C07209=1031.022,-23.750,-88.174,168.001,42.640,157.928
C07210=1031.029,-23.500,-88.188,168.003,42.639,157.928
C07211=1031.035,-23.251,-88.201,168.006,42.638,157.928
C07212=1031.041,-23.002,-88.215,168.009,42.636,157.928
C07213=1031.047,-22.752,-88.229,168.012,42.635,157.928
C07214=1031.053,-22.502,-88.242,168.014,42.634,157.928
C07215=1031.060,-22.253,-88.255,168.016,42.633,157.928
C07216=1031.066,-22.003,-88.270,168.019,42.631,157.928
C07217=1031.072,-21.754,-88.283,168.022,42.630,157.928
C07218=1031.078,-21.504,-88.296,168.025,42.629,157.928
C07219=1031.084,-21.254,-88.310,168.026,42.627,157.928
C07220=1031.091,-21.005,-88.324,168.029,42.626,157.928
C07221=1031.097,-20.756,-88.338,168.032,42.625,157.928
C07222=1031.104,-20.474,-88.353,168.035,42.623,157.928
C07223=1031.111,-20.193,-88.369,168.038,42.622,157.928
C07224=1031.118,-19.911,-88.384,168.040,42.621,157.928
C07225=1031.125,-19.630,-88.399,168.043,42.619,157.928
C07226=1031.131,-19.380,-88.413,168.046,42.618,157.928
C07227=1031.138,-19.130,-88.426,168.049,42.617,157.928
C07228=1031.145,-18.881,-88.441,168.051,42.615,157.927
C07229=1031.150,-18.632,-88.455,168.053,42.614,157.927
C07230=1031.156,-18.382,-88.468,168.056,42.613,157.927
C07231=1031.163,-18.132,-88.481,168.059,42.611,157.927
C07232=1031.169,-17.883,-88.495,168.061,42.610,157.927
C07233=1031.176,-17.633,-88.510,168.064,42.609,157.927
C07234=1031.182,-17.384,-88.523,168.066,42.608,157.927
C07235=1031.188,-17.134,-88.537,168.069,42.606,157.927
C07236=1031.194,-16.885,-88.550,168.071,42.605,157.927
C07237=1031.200,-16.635,-88.564,168.074,42.604,157.927
C07238=1031.207,-16.386,-88.579,168.077,42.602,157.927
C07239=1031.213,-16.136,-88.592,168.079,42.601,157.927
C07240=1031.220,-15.886,-88.606,168.081,42.600,157.927
C07241=1031.226,-15.638,-88.620,168.084,42.598,157.927
C07242=1031.232,-15.388,-88.634,168.087,42.597,157.927
C07243=1031.238,-15.138,-88.648,168.090,42.596,157.927
C07244=1031.245,-14.889,-88.662,168.091,42.595,157.927
C07245=1031.251,-14.639,-88.676,168.094,42.594,157.927
C07246=1031.257,-14.389,-88.690,168.097,42.592,157.927
C07247=1031.263,-14.140,-88.704,168.099,42.591,157.926
C07248=1031.269,-13.890,-88.718,168.102,42.590,157.926
C07249=1031.275,-13.641,-88.732,168.105,42.589,157.926
C07250=1031.282,-13.391,-88.747,168.106,42.588,157.926
C07251=1031.288,-13.142,-88.760,168.109,42.586,157.926
C07252=1031.294,-12.892,-88.775,168.112,42.585,157.926
C07253=1031.300,-12.642,-88.789,168.114,42.584,157.926
C07254=1031.307,-12.393,-88.803,168.117,42.583,157.926
C07255=1031.313,-12.144,-88.817,168.119,42.581,157.926
C07256=1031.319,-11.894,-88.830,168.121,42.580,157.926
C07257=1031.325,-11.645,-88.845,168.124,42.579,157.926
C07258=1031.332,-11.395,-88.859,168.127,42.578,157.926
C07259=1031.338,-11.146,-88.873,168.130,42.576,157.926
C07260=1031.344,-10.895,-88.888,168.132,42.575,157.926
C07261=1031.350,-10.647,-88.901,168.134,42.574,157.926
C07262=1031.356,-10.396,-88.916,168.137,42.573,157.926
C07263=1031.363,-10.148,-88.930,168.139,42.572,157.926
C07264=1031.369,-9.898,-88.944,168.142,42.570,157.926
C07265=1031.375,-9.648,-88.959,168.145,42.569,157.926
C07266=1031.382,-9.399,-88.972,168.146,42.568,157.926
C07267=1031.388,-9.149,-88.987,168.149,42.567,157.926
C07268=1031.394,-8.900,-89.002,168.152,42.566,157.926
C07269=1031.401,-8.650,-89.015,168.154,42.564,157.925
C07270=1031.406,-8.401,-89.030,168.157,42.563,157.925
C07271=1031.413,-8.151,-89.044,168.160,42.562,157.925
C07272=1031.420,-7.901,-89.058,168.161,42.561,157.925
C07273=1031.425,-7.652,-89.072,168.164,42.559,157.925
C07274=1031.432,-7.403,-89.087,168.167,42.558,157.925
C07275=1031.438,-7.154,-89.101,168.169,42.557,157.925
C07276=1031.445,-6.904,-89.115,168.172,42.556,157.925
C07277=1031.451,-6.654,-89.130,168.175,42.555,157.925
C07278=1031.457,-6.404,-89.144,168.176,42.553,157.925
C07279=1031.464,-6.155,-89.158,168.179,42.552,157.925
C07280=1031.470,-5.905,-89.173,168.182,42.551,157.925
C07281=1031.476,-5.656,-89.187,168.184,42.550,157.925
C07282=1031.483,-5.406,-89.201,168.186,42.548,157.925
C07283=1031.489,-5.157,-89.216,168.189,42.547,157.925
C07284=1031.495,-4.908,-89.229,168.191,42.546,157.925
C07285=1031.502,-4.658,-89.244,168.194,42.545,157.925
C07286=1031.509,-4.374,-89.261,168.197,42.543,157.925
C07287=1031.516,-4.092,-89.277,168.199,42.542,157.925
C07288=1031.523,-3.809,-89.293,168.202,42.540,157.924
C07289=1031.530,-3.526,-89.310,168.205,42.539,157.924
C07290=1031.537,-3.276,-89.325,168.208,42.538,157.924
C07291=1031.543,-3.027,-89.339,168.210,42.537,157.924
C07292=1031.549,-2.777,-89.354,168.213,42.536,157.924
C07293=1031.555,-2.528,-89.369,168.215,42.535,157.924
C07294=1031.561,-2.278,-89.383,168.217,42.534,157.924
C07295=1031.567,-2.028,-89.398,168.220,42.533,157.924
C07296=1031.574,-1.779,-89.413,168.222,42.532,157.924
C07297=1031.579,-1.530,-89.427,168.225,42.531,157.924
C07298=1031.586,-1.280,-89.442,168.227,42.530,157.924
C07299=1031.592,-1.031,-89.457,168.230,42.529,157.924
C07300=1031.598,-0.782,-89.472,168.232,42.527,157.924
C07301=1031.604,-0.532,-89.487,168.234,42.527,157.924
C07302=1031.610,-0.282,-89.501,168.237,42.525,157.924
C07303=1031.616,-0.033,-89.516,168.239,42.524,157.924
C07304=1031.623,0.217,-89.530,168.242,42.523,157.924
C07305=1031.629,0.467,-89.545,168.245,42.522,157.924
C07306=1031.635,0.716,-89.560,168.246,42.521,157.924
C07307=1031.641,0.965,-89.575,168.249,42.519,157.924
C07308=1031.647,1.215,-89.590,168.251,42.518,157.924
C07309=1031.654,1.465,-89.605,168.254,42.517,157.924
C07310=1031.660,1.713,-89.619,168.257,42.516,157.924
C07311=1031.666,1.963,-89.634,168.259,42.515,157.924
C07312=1031.672,2.213,-89.649,168.261,42.514,157.924
C07313=1031.679,2.462,-89.664,168.263,42.513,157.924
C07314=1031.685,2.711,-89.679,168.266,42.512,157.924
C07315=1031.691,2.961,-89.694,168.268,42.511,157.924
C07316=1031.697,3.211,-89.709,168.271,42.510,157.924
C07317=1031.704,3.460,-89.724,168.274,42.509,157.924
C07318=1031.710,3.709,-89.738,168.275,42.507,157.923
C07319=1031.716,3.959,-89.753,168.278,42.506,157.923
C07320=1031.722,4.209,-89.768,168.280,42.505,157.923
C07321=1031.729,4.458,-89.783,168.283,42.504,157.923
C07322=1031.734,4.707,-89.798,168.286,42.503,157.923
C07323=1031.741,4.957,-89.813,168.288,42.502,157.923
C07324=1031.747,5.207,-89.828,168.290,42.501,157.923
C07325=1031.754,5.456,-89.843,168.292,42.500,157.923
C07326=1031.760,5.706,-89.857,168.295,42.499,157.923
C07327=1031.766,5.956,-89.872,168.298,42.497,157.923
C07328=1031.772,6.204,-89.888,168.300,42.496,157.923
C07329=1031.779,6.454,-89.903,168.303,42.495,157.923
C07330=1031.785,6.703,-89.918,168.304,42.494,157.923
C07331=1031.792,6.953,-89.933,168.307,42.493,157.923
C07332=1031.798,7.203,-89.947,168.309,42.492,157.923
C07333=1031.804,7.452,-89.962,168.312,42.491,157.923
C07334=1031.810,7.701,-89.977,168.315,42.489,157.923
C07335=1031.817,7.951,-89.992,168.316,42.488,157.923
C07336=1031.823,8.200,-90.008,168.319,42.487,157.923
C07337=1031.830,8.449,-90.023,168.321,42.486,157.923
C07338=1031.836,8.699,-90.038,168.324,42.485,157.923
C07339=1031.842,8.949,-90.052,168.327,42.483,157.923
C07340=1031.849,9.198,-90.067,168.329,42.482,157.923
C07341=1031.855,9.447,-90.083,168.332,42.481,157.923
C07342=1031.861,9.696,-90.098,168.333,42.480,157.922
C07343=1031.868,9.946,-90.113,168.336,42.479,157.922
C07344=1031.874,10.196,-90.128,168.338,42.478,157.922
C07345=1031.880,10.445,-90.142,168.341,42.477,157.922
C07346=1031.887,10.694,-90.158,168.344,42.475,157.922
C07347=1031.893,10.944,-90.173,168.345,42.474,157.922
C07348=1031.900,11.194,-90.188,168.348,42.473,157.922
C07349=1031.906,11.443,-90.203,168.350,42.472,157.922
C07350=1031.913,11.728,-90.220,168.353,42.471,157.922
C07351=1031.921,12.013,-90.238,168.356,42.469,157.922
C07352=1031.928,12.298,-90.256,168.358,42.468,157.922
C07353=1031.935,12.583,-90.272,168.361,42.467,157.922
C07354=1031.942,12.833,-90.288,168.364,42.465,157.922
C07355=1031.948,13.082,-90.303,168.366,42.464,157.922
C07356=1031.954,13.332,-90.318,168.369,42.463,157.922
C07357=1031.961,13.581,-90.333,168.370,42.462,157.922
C07358=1031.967,13.831,-90.348,168.373,42.461,157.922
C07359=1031.974,14.080,-90.363,168.376,42.459,157.922
C07360=1031.980,14.330,-90.380,168.378,42.458,157.922
C07361=1031.986,14.579,-90.395,168.381,42.457,157.922
C07362=1031.993,14.828,-90.410,168.383,42.456,157.922
C07363=1031.998,15.078,-90.426,168.386,42.455,157.922
C07364=1032.005,15.328,-90.441,168.387,42.454,157.922
C07365=1032.012,15.577,-90.456,168.390,42.453,157.921
C07366=1032.017,15.827,-90.472,168.392,42.452,157.921
C07367=1032.024,16.076,-90.488,168.395,42.451,157.921
C07368=1032.030,16.326,-90.503,168.397,42.450,157.921
C07369=1032.037,16.575,-90.518,168.400,42.448,157.921
C07370=1032.043,16.825,-90.534,168.401,42.447,157.921
C07371=1032.049,17.073,-90.549,168.404,42.446,157.921
C07372=1032.055,17.323,-90.564,168.406,42.445,157.921
C07373=1032.061,17.572,-90.580,168.409,42.444,157.921
C07374=1032.067,17.822,-90.595,168.411,42.443,157.921
C07375=1032.074,18.071,-90.611,168.414,42.442,157.921
C07376=1032.080,18.321,-90.627,168.415,42.441,157.921
C07377=1032.087,18.570,-90.642,168.418,42.440,157.921
C07378=1032.093,18.820,-90.657,168.420,42.439,157.921
C07379=1032.099,19.069,-90.674,168.423,42.438,157.921
C07380=1032.106,19.319,-90.689,168.426,42.437,157.921
C07381=1032.112,19.568,-90.704,168.428,42.436,157.921
C07382=1032.118,19.817,-90.720,168.431,42.435,157.921
C07383=1032.125,20.067,-90.735,168.432,42.434,157.921
C07384=1032.131,20.316,-90.752,168.435,42.433,157.921
C07385=1032.137,20.566,-90.767,168.437,42.432,157.921
C07386=1032.143,20.815,-90.783,168.440,42.431,157.921
C07387=1032.150,21.064,-90.799,168.442,42.430,157.921
C07388=1032.156,21.314,-90.813,168.445,42.428,157.921
C07389=1032.162,21.563,-90.830,168.446,42.427,157.920
C07390=1032.169,21.812,-90.845,168.448,42.426,157.920
C07391=1032.174,22.062,-90.861,168.451,42.425,157.920
C07392=1032.181,22.311,-90.877,168.453,42.424,157.920
C07393=1032.187,22.561,-90.893,168.456,42.423,157.920
C07394=1032.193,22.810,-90.908,168.458,42.422,157.920
C07395=1032.199,23.060,-90.924,168.460,42.421,157.920
C07396=1032.206,23.309,-90.940,168.462,42.420,157.920
C07397=1032.213,23.559,-90.956,168.465,42.418,157.920
C07398=1032.219,23.809,-90.971,168.467,42.418,157.920
C07399=1032.225,24.058,-90.988,168.470,42.416,157.920
C07400=1032.232,24.307,-91.003,168.472,42.415,157.920
C07401=1032.237,24.557,-91.019,168.475,42.414,157.920
C07402=1032.244,24.806,-91.034,168.476,42.413,157.920
C07403=1032.250,25.055,-91.051,168.479,42.412,157.920
C07404=1032.257,25.304,-91.066,168.481,42.411,157.920
C07405=1032.263,25.554,-91.083,168.484,42.410,157.920
C07406=1032.270,25.804,-91.098,168.486,42.409,157.920
C07407=1032.275,26.053,-91.114,168.489,42.408,157.920
C07408=1032.282,26.302,-91.130,168.490,42.407,157.920
C07409=1032.288,26.552,-91.146,168.493,42.406,157.920
C07410=1032.295,26.801,-91.162,168.495,42.405,157.920
C07411=1032.300,27.051,-91.177,168.498,42.404,157.920
C07412=1032.307,27.300,-91.193,168.500,42.403,157.920
C07413=1032.314,27.550,-91.210,168.503,42.401,157.920
C07414=1032.320,27.835,-91.228,168.505,42.400,157.920
C07415=1032.328,28.122,-91.246,168.507,42.399,157.919
C07416=1032.335,28.409,-91.264,168.510,42.398,157.919
C07417=1032.342,28.695,-91.283,168.513,42.397,157.919
C07418=1032.348,28.944,-91.299,168.516,42.396,157.919
C07419=1032.355,29.193,-91.315,168.518,42.395,157.919
C07420=1032.361,29.442,-91.331,168.520,42.394,157.919
C07421=1032.367,29.692,-91.347,168.522,42.393,157.919
C07422=1032.374,29.942,-91.364,168.524,42.392,157.919
C07423=1032.380,30.191,-91.380,168.527,42.391,157.919
C07424=1032.386,30.440,-91.396,168.529,42.390,157.919
C07425=1032.392,30.690,-91.412,168.532,42.389,157.919
C07426=1032.399,30.939,-91.428,168.534,42.388,157.919
C07427=1032.405,31.189,-91.445,168.536,42.386,157.919
C07428=1032.411,31.438,-91.461,168.538,42.386,157.919
C07429=1032.418,31.687,-91.476,168.540,42.385,157.919
C07430=1032.424,31.936,-91.493,168.543,42.383,157.919
C07431=1032.430,32.186,-91.509,168.545,42.382,157.919
C07432=1032.436,32.436,-91.526,168.548,42.381,157.919
C07433=1032.443,32.685,-91.541,168.550,42.380,157.919
C07434=1032.449,32.934,-91.558,168.552,42.379,157.919
C07435=1032.455,33.184,-91.574,168.554,42.378,157.919
C07436=1032.461,33.433,-91.590,168.557,42.377,157.919
C07437=1032.468,33.683,-91.606,168.559,42.376,157.919
C07438=1032.474,33.932,-91.622,168.562,42.375,157.919
C07439=1032.480,34.181,-91.639,168.564,42.374,157.919
C07440=1032.487,34.430,-91.654,168.566,42.373,157.919
C07441=1032.493,34.680,-91.671,168.568,42.372,157.919
C07442=1032.499,34.930,-91.687,168.570,42.371,157.919
C07443=1032.506,35.179,-91.704,168.573,42.370,157.919
C07444=1032.512,35.428,-91.720,168.575,42.369,157.918
C07445=1032.519,35.678,-91.736,168.578,42.368,157.918
C07446=1032.525,35.927,-91.753,168.580,42.367,157.918
C07447=1032.531,36.176,-91.769,168.582,42.366,157.918
C07448=1032.538,36.426,-91.785,168.584,42.365,157.918
C07449=1032.544,36.675,-91.801,168.587,42.364,157.918
C07450=1032.550,36.924,-91.818,168.589,42.363,157.918
C07451=1032.556,37.173,-91.834,168.591,42.362,157.918
C07452=1032.563,37.424,-91.851,168.594,42.361,157.918
C07453=1032.569,37.673,-91.867,168.596,42.360,157.918
C07454=1032.575,37.922,-91.884,168.598,42.359,157.918
C07455=1032.581,38.172,-91.901,168.600,42.358,157.918
C07456=1032.587,38.421,-91.917,168.603,42.357,157.918
C07457=1032.593,38.670,-91.933,168.605,42.356,157.918
C07458=1032.599,38.920,-91.950,168.607,42.355,157.918
C07459=1032.607,39.169,-91.966,168.610,42.354,157.918
C07460=1032.613,39.418,-91.983,168.612,42.353,157.918
C07461=1032.619,39.668,-91.999,168.615,42.352,157.918
C07462=1032.626,39.917,-92.016,168.616,42.351,157.918
C07463=1032.632,40.166,-92.033,168.618,42.350,157.918
C07464=1032.638,40.416,-92.049,168.621,42.349,157.918
C07465=1032.644,40.665,-92.066,168.623,42.348,157.918
C07466=1032.653,41.053,-92.091,168.627,42.347,157.918
C07467=1032.663,41.442,-92.117,168.631,42.345,157.918
C07468=1032.673,41.830,-92.144,168.634,42.344,157.918
C07469=1032.684,42.219,-92.169,168.637,42.342,157.918
C07470=1032.690,42.467,-92.186,168.640,42.341,157.918
C07471=1032.696,42.717,-92.203,168.642,42.340,157.918
C07472=1032.702,42.967,-92.219,168.645,42.339,157.918
C07473=1032.708,43.216,-92.237,168.646,42.338,157.917
C07474=1032.717,43.613,-92.263,168.650,42.337,157.918
C07475=1032.727,44.009,-92.290,168.653,42.335,157.917
C07476=1032.737,44.406,-92.317,168.657,42.334,157.918
C07477=1032.747,44.803,-92.344,168.661,42.332,157.917
C07478=1032.753,45.051,-92.361,168.663,42.331,157.917
C07479=1032.760,45.301,-92.377,168.666,42.331,157.917
C07480=1032.765,45.550,-92.395,168.667,42.330,157.917
C07481=1032.772,45.800,-92.412,168.669,42.329,157.917
C07482=1032.778,46.049,-92.429,168.672,42.328,157.917
C07483=1032.784,46.298,-92.445,168.674,42.327,157.917
C07484=1032.790,46.548,-92.463,168.677,42.326,157.917
C07485=1032.796,46.798,-92.479,168.679,42.326,157.917
C07486=1032.802,47.046,-92.496,168.681,42.325,157.917
C07487=1032.809,47.296,-92.513,168.684,42.323,157.917
C07488=1032.814,47.545,-92.530,168.685,42.322,157.917
C07489=1032.821,47.795,-92.548,168.687,42.322,157.917
C07490=1032.827,48.044,-92.564,168.690,42.320,157.917
C07491=1032.834,48.294,-92.581,168.692,42.319,157.917
C07492=1032.839,48.543,-92.599,168.695,42.319,157.917
C07493=1032.845,48.792,-92.615,168.697,42.318,157.917
C07494=1032.852,49.041,-92.632,168.699,42.317,157.917
C07495=1032.858,49.290,-92.650,168.702,42.316,157.917
C07496=1032.864,49.541,-92.667,168.703,42.315,157.917
C07497=1032.871,49.789,-92.684,168.705,42.314,157.917
C07498=1032.877,50.039,-92.701,168.708,42.313,157.917
C07499=1032.883,50.288,-92.718,168.710,42.313,157.917
C07500=1032.889,50.537,-92.735,168.713,42.312,157.917
C07501=1032.896,50.786,-92.752,168.715,42.311,157.917
C07502=1032.902,51.036,-92.768,168.717,42.310,157.917
C07503=1032.908,51.286,-92.786,168.720,42.309,157.917
C07504=1032.914,51.534,-92.803,168.721,42.308,157.917
C07505=1032.921,51.784,-92.820,168.724,42.306,157.917
C07506=1032.926,52.033,-92.837,168.726,42.306,157.917
C07507=1032.933,52.283,-92.855,168.728,42.305,157.917
C07508=1032.939,52.532,-92.872,168.731,42.303,157.917
C07509=1032.946,52.782,-92.888,168.733,42.303,157.917
C07510=1032.951,53.031,-92.906,168.735,42.302,157.917
C07511=1032.958,53.280,-92.923,168.738,42.301,157.917
C07512=1032.964,53.529,-92.940,168.739,42.300,157.917
C07513=1032.970,53.779,-92.957,168.742,42.299,157.917
C07514=1032.977,54.028,-92.974,168.744,42.298,157.917
C07515=1032.983,54.277,-92.992,168.746,42.297,157.917
C07516=1032.989,54.526,-93.009,168.749,42.296,157.916
C07517=1032.996,54.776,-93.027,168.751,42.295,157.916
C07518=1033.002,55.026,-93.043,168.753,42.294,157.916
C07519=1033.009,55.275,-93.060,168.755,42.293,157.916
C07520=1033.015,55.524,-93.078,168.757,42.292,157.916
C07521=1033.021,55.773,-93.095,168.760,42.291,157.916
C07522=1033.028,56.022,-93.112,168.762,42.290,157.916
C07523=1033.033,56.272,-93.129,168.765,42.290,157.916
C07524=1033.040,56.522,-93.147,168.767,42.289,157.916
C07525=1033.047,56.771,-93.164,168.769,42.288,157.916
C07526=1033.052,57.020,-93.182,168.771,42.287,157.916
C07527=1033.059,57.269,-93.199,168.773,42.286,157.916
C07528=1033.065,57.518,-93.216,168.776,42.284,157.916
C07529=1033.071,57.768,-93.234,168.778,42.284,157.916
C07530=1033.078,58.017,-93.251,168.780,42.283,157.916
C07531=1033.084,58.267,-93.267,168.783,42.281,157.916
C07532=1033.090,58.516,-93.285,168.785,42.280,157.916
C07533=1033.097,58.765,-93.302,168.787,42.279,157.916
C07534=1033.104,59.015,-93.320,168.789,42.278,157.916
C07535=1033.110,59.264,-93.338,168.791,42.277,157.916
C07536=1033.116,59.513,-93.355,168.794,42.276,157.916
C07537=1033.123,59.763,-93.372,168.796,42.275,157.916
C07538=1033.130,60.048,-93.392,168.799,42.274,157.916
C07539=1033.137,60.334,-93.412,168.802,42.273,157.916
C07540=1033.144,60.620,-93.431,168.803,42.272,157.916
C07541=1033.152,60.907,-93.451,168.806,42.270,157.915
C07542=1033.158,61.155,-93.468,168.809,42.269,157.915
C07543=1033.164,61.405,-93.486,168.811,42.268,157.915
C07544=1033.171,61.655,-93.504,168.813,42.267,157.915
C07545=1033.177,61.903,-93.521,168.815,42.266,157.915
C07546=1033.184,62.153,-93.539,168.817,42.265,157.915
C07547=1033.190,62.402,-93.556,168.820,42.264,157.915
C07548=1033.197,62.651,-93.573,168.822,42.263,157.915
C07549=1033.203,62.901,-93.591,168.824,42.262,157.915
C07550=1033.210,63.150,-93.608,168.827,42.261,157.915
C07551=1033.216,63.399,-93.625,168.829,42.260,157.915
C07552=1033.222,63.649,-93.643,168.831,42.259,157.915
C07553=1033.228,63.898,-93.662,168.833,42.259,157.915
C07554=1033.235,64.147,-93.679,168.835,42.258,157.915
C07555=1033.241,64.396,-93.697,168.838,42.257,157.915
C07556=1033.248,64.646,-93.714,168.840,42.256,157.915
C07557=1033.253,64.895,-93.732,168.843,42.255,157.915
C07558=1033.259,65.145,-93.749,168.845,42.254,157.915
C07559=1033.266,65.394,-93.767,168.846,42.253,157.915
C07560=1033.273,65.643,-93.785,168.849,42.252,157.915
C07561=1033.279,65.892,-93.802,168.851,42.252,157.915
C07562=1033.285,66.142,-93.820,168.853,42.251,157.915
C07563=1033.291,66.391,-93.838,168.856,42.249,157.915
C07564=1033.297,66.640,-93.855,168.858,42.249,157.915
C07565=1033.304,66.889,-93.874,168.860,42.248,157.915
C07566=1033.310,67.139,-93.892,168.863,42.246,157.915
C07567=1033.316,67.388,-93.909,168.864,42.246,157.915
C07568=1033.322,67.637,-93.927,168.867,42.244,157.915
C07569=1033.329,67.887,-93.945,168.869,42.244,157.915
C07570=1033.336,68.136,-93.963,168.871,42.243,157.915
C07571=1033.341,68.385,-93.980,168.874,42.242,157.915
C07572=1033.347,68.635,-93.998,168.876,42.241,157.915
C07573=1033.354,68.884,-94.017,168.878,42.240,157.915
C07574=1033.360,69.133,-94.034,168.881,42.239,157.914
C07575=1033.366,69.382,-94.052,168.882,42.238,157.914
C07576=1033.372,69.631,-94.070,168.884,42.238,157.915
C07577=1033.379,69.881,-94.088,168.887,42.237,157.914
C07578=1033.385,70.130,-94.105,168.889,42.236,157.914
C07579=1033.391,70.379,-94.124,168.892,42.235,157.914
C07580=1033.397,70.629,-94.142,168.894,42.234,157.914
C07581=1033.403,70.879,-94.160,168.896,42.233,157.914
C07582=1033.409,71.127,-94.178,168.899,42.232,157.914
C07583=1033.415,71.377,-94.196,168.901,42.231,157.914
C07584=1033.423,71.626,-94.214,168.902,42.230,157.914
C07585=1033.429,71.875,-94.232,168.905,42.229,157.914
C07586=1033.434,72.124,-94.250,168.907,42.228,157.914
C07587=1033.441,72.373,-94.268,168.909,42.228,157.914
C07588=1033.447,72.623,-94.286,168.912,42.227,157.914
C07589=1033.453,72.872,-94.305,168.914,42.226,157.914
C07590=1033.460,73.122,-94.322,168.916,42.225,157.914
C07591=1033.466,73.370,-94.340,168.919,42.224,157.914
C07592=1033.472,73.620,-94.358,168.921,42.224,157.914
C07593=1033.478,73.869,-94.377,168.922,42.223,157.914
C07594=1033.485,74.119,-94.395,168.925,42.222,157.914
C07595=1033.491,74.368,-94.414,168.927,42.221,157.914
C07596=1033.496,74.617,-94.431,168.930,42.220,157.914
C07597=1033.503,74.866,-94.450,168.932,42.219,157.914
C07598=1033.510,75.115,-94.467,168.934,42.218,157.914
C07599=1033.516,75.365,-94.486,168.937,42.217,157.914
C07600=1033.522,75.614,-94.504,168.939,42.216,157.914
C07601=1033.528,75.863,-94.522,168.940,42.215,157.914
C07602=1033.536,76.149,-94.542,168.943,42.214,157.914
C07603=1033.542,76.435,-94.564,168.946,42.213,157.914
C07604=1033.550,76.721,-94.585,168.948,42.212,157.914
C07605=1033.557,77.006,-94.605,168.951,42.211,157.914
C07606=1033.564,77.255,-94.624,168.954,42.210,157.914
C07607=1033.570,77.505,-94.642,168.956,42.209,157.914
C07608=1033.576,77.754,-94.660,168.958,42.209,157.914
C07609=1033.582,78.003,-94.678,168.960,42.208,157.914
C07610=1033.588,78.252,-94.697,168.962,42.207,157.914
C07611=1033.595,78.502,-94.715,168.964,42.206,157.914
C07612=1033.600,78.752,-94.734,168.967,42.205,157.914
C07613=1033.607,79.001,-94.753,168.969,42.204,157.914
C07614=1033.613,79.250,-94.771,168.971,42.203,157.914
C07615=1033.618,79.499,-94.789,168.974,42.202,157.914
C07616=1033.625,79.748,-94.807,168.976,42.202,157.914
C07617=1033.631,79.997,-94.826,168.978,42.201,157.914
C07618=1033.638,80.246,-94.845,168.980,42.200,157.914
C07619=1033.643,80.496,-94.863,168.982,42.199,157.914
C07620=1033.650,80.745,-94.882,168.984,42.199,157.914
C07621=1033.656,80.995,-94.901,168.987,42.198,157.914
C07622=1033.662,81.244,-94.918,168.989,42.197,157.914
C07623=1033.668,81.493,-94.937,168.991,42.196,157.914
C07624=1033.674,81.742,-94.955,168.994,42.195,157.914
C07625=1033.681,81.991,-94.974,168.996,42.194,157.914
C07626=1033.686,82.240,-94.993,168.998,42.193,157.913
C07627=1033.693,82.490,-95.011,169.000,42.192,157.913
C07628=1033.699,82.739,-95.030,169.002,42.192,157.914
C07629=1033.705,82.988,-95.049,169.004,42.191,157.913
C07630=1033.712,83.238,-95.067,169.007,42.190,157.913
C07631=1033.718,83.487,-95.086,169.009,42.189,157.913
C07632=1033.724,83.736,-95.103,169.011,42.188,157.913
C07633=1033.730,83.985,-95.123,169.014,42.188,157.913
C07634=1033.736,84.234,-95.141,169.016,42.187,157.913
C07635=1033.742,84.483,-95.160,169.018,42.186,157.913
C07636=1033.749,84.732,-95.179,169.020,42.185,157.913
C07637=1033.755,84.982,-95.197,169.022,42.184,157.913
C07638=1033.761,85.231,-95.215,169.025,42.183,157.913
C07639=1033.767,85.481,-95.234,169.027,42.182,157.913
C07640=1033.773,85.730,-95.253,169.029,42.181,157.913
C07641=1033.780,85.979,-95.272,169.032,42.180,157.913
C07642=1033.786,86.228,-95.290,169.034,42.180,157.913
C07643=1033.793,86.477,-95.309,169.036,42.179,157.913
C07644=1033.799,86.726,-95.328,169.039,42.178,157.913
C07645=1033.805,86.976,-95.347,169.040,42.177,157.913
C07646=1033.811,87.226,-95.365,169.042,42.176,157.913
C07647=1033.817,87.475,-95.384,169.045,42.176,157.913
C07648=1033.824,87.724,-95.402,169.047,42.175,157.913
C07649=1033.830,87.973,-95.421,169.050,42.173,157.913
C07650=1033.837,88.222,-95.439,169.052,42.173,157.913
C07651=1033.842,88.472,-95.459,169.054,42.172,157.913
C07652=1033.849,88.721,-95.477,169.057,42.171,157.913
C07653=1033.855,88.970,-95.496,169.059,42.170,157.913
C07654=1033.862,89.219,-95.515,169.060,42.169,157.913
C07655=1033.868,89.468,-95.533,169.063,42.168,157.913
C07656=1033.874,89.717,-95.552,169.065,42.167,157.913
C07657=1033.880,89.967,-95.571,169.068,42.166,157.913
C07658=1033.887,90.216,-95.590,169.070,42.166,157.913
C07659=1033.892,90.465,-95.609,169.072,42.165,157.913
C07660=1033.899,90.714,-95.628,169.075,42.164,157.913
C07661=1033.904,90.964,-95.647,169.077,42.164,157.913
C07662=1033.911,91.212,-95.666,169.079,42.163,157.913
C07663=1033.918,91.461,-95.685,169.081,42.161,157.913
C07664=1033.923,91.711,-95.704,169.083,42.161,157.913
C07665=1033.930,91.960,-95.723,169.085,42.160,157.913
C07666=1033.937,92.246,-95.745,169.088,42.159,157.913
C07667=1033.944,92.531,-95.767,169.091,42.158,157.913
C07668=1033.951,92.817,-95.788,169.093,42.157,157.913
C07669=1033.958,93.102,-95.810,169.096,42.157,157.913
C07670=1033.963,93.352,-95.829,169.098,42.156,157.913
C07671=1033.970,93.601,-95.848,169.101,42.155,157.913
C07672=1033.976,93.851,-95.868,169.103,42.154,157.913
C07673=1033.983,94.100,-95.887,169.104,42.153,157.913
C07674=1033.988,94.349,-95.906,169.107,42.152,157.913
C07675=1033.995,94.598,-95.925,169.109,42.151,157.913
C07676=1034.001,94.848,-95.944,169.112,42.151,157.913
C07677=1034.007,95.096,-95.963,169.114,42.150,157.913
C07678=1034.013,95.346,-95.983,169.116,42.149,157.913
C07679=1034.019,95.595,-96.001,169.119,42.149,157.913
C07680=1034.025,95.844,-96.021,169.121,42.148,157.913
C07681=1034.032,96.093,-96.039,169.123,42.147,157.913
C07682=1034.038,96.342,-96.059,169.125,42.146,157.913
C07683=1034.044,96.591,-96.078,169.128,42.145,157.913
C07684=1034.051,96.841,-96.097,169.129,42.144,157.913
C07685=1034.057,97.090,-96.117,169.132,42.143,157.913
C07686=1034.063,97.339,-96.135,169.134,42.142,157.913
C07687=1034.069,97.588,-96.155,169.137,42.142,157.913
C07688=1034.075,97.838,-96.173,169.139,42.141,157.913
C07689=1034.081,98.086,-96.193,169.141,42.140,157.913
C07690=1034.088,98.335,-96.212,169.144,42.139,157.913
C07691=1034.094,98.585,-96.231,169.146,42.139,157.913
C07692=1034.101,98.834,-96.251,169.148,42.138,157.913
C07693=1034.107,99.084,-96.270,169.150,42.137,157.913
C07694=1034.113,99.333,-96.289,169.152,42.136,157.913
C07695=1034.119,99.581,-96.309,169.155,42.135,157.913
C07696=1034.125,99.831,-96.327,169.157,42.134,157.913
C07697=1034.131,100.080,-96.347,169.159,42.133,157.913
C07698=1034.138,100.330,-96.367,169.162,42.133,157.913
C07699=1034.144,100.579,-96.386,169.164,42.132,157.913
C07700=1034.150,100.827,-96.406,169.166,42.131,157.912
C07701=1034.156,101.077,-96.425,169.169,42.131,157.913
C07702=1034.162,101.326,-96.445,169.171,42.130,157.913
C07703=1034.168,101.575,-96.463,169.173,42.128,157.913
C07704=1034.175,101.825,-96.483,169.175,42.128,157.913
C07705=1034.181,102.074,-96.503,169.177,42.127,157.913
C07706=1034.186,102.323,-96.522,169.180,42.127,157.913
C07707=1034.193,102.572,-96.542,169.182,42.126,157.913
C07708=1034.199,102.821,-96.561,169.184,42.125,157.913
C07709=1034.205,103.070,-96.581,169.187,42.124,157.913
C07710=1034.211,103.319,-96.601,169.189,42.124,157.913
C07711=1034.217,103.569,-96.620,169.191,42.123,157.913
C07712=1034.224,103.817,-96.640,169.194,42.122,157.913
C07713=1034.229,104.067,-96.659,169.196,42.121,157.913
C07714=1034.235,104.316,-96.679,169.197,42.120,157.912
C07715=1034.242,104.566,-96.699,169.201,42.120,157.913
C07716=1034.248,104.814,-96.718,169.202,42.119,157.913
C07717=1034.254,105.064,-96.737,169.205,42.118,157.913
C07718=1034.260,105.313,-96.757,169.207,42.118,157.913
C07719=1034.266,105.561,-96.777,169.209,42.117,157.913
C07720=1034.272,105.811,-96.797,169.212,42.116,157.913
C07721=1034.279,106.060,-96.816,169.214,42.115,157.913
C07722=1034.285,106.309,-96.835,169.217,42.114,157.913
C07723=1034.291,106.558,-96.855,169.219,42.114,157.913
C07724=1034.297,106.808,-96.876,169.221,42.113,157.913
C07725=1034.304,107.057,-96.894,169.224,42.112,157.913
C07726=1034.310,107.306,-96.914,169.226,42.111,157.913
C07727=1034.316,107.554,-96.934,169.227,42.111,157.913
C07728=1034.322,107.805,-96.954,169.230,42.109,157.913
C07729=1034.328,108.053,-96.974,169.232,42.109,157.913
C07730=1034.335,108.339,-96.996,169.235,42.108,157.913
C07731=1034.343,108.625,-97.018,169.238,42.107,157.913
C07732=1034.349,108.910,-97.041,169.241,42.106,157.913
C07733=1034.356,109.196,-97.063,169.243,42.106,157.913
C07734=1034.363,109.445,-97.084,169.246,42.105,157.913
C07735=1034.369,109.694,-97.104,169.248,42.104,157.912
C07736=1034.376,109.943,-97.123,169.250,42.102,157.912
C07737=1034.382,110.193,-97.143,169.252,42.102,157.913
C07738=1034.388,110.442,-97.163,169.254,42.101,157.912
C07739=1034.394,110.690,-97.183,169.257,42.101,157.913
C07740=1034.400,110.939,-97.203,169.259,42.100,157.913
C07741=1034.406,111.189,-97.222,169.261,42.099,157.912
C07742=1034.412,111.438,-97.242,169.264,42.098,157.913
C07743=1034.418,111.687,-97.262,169.266,42.098,157.913
C07744=1034.425,111.937,-97.282,169.269,42.096,157.912
C07745=1034.431,112.185,-97.302,169.271,42.096,157.913
C07746=1034.437,112.434,-97.322,169.273,42.095,157.912
C07747=1034.443,112.684,-97.342,169.276,42.095,157.913
C07748=1034.449,112.933,-97.362,169.278,42.094,157.913
C07749=1034.455,113.182,-97.382,169.280,42.093,157.913
C07750=1034.462,113.431,-97.402,169.282,42.092,157.913
C07751=1034.468,113.680,-97.422,169.284,42.092,157.913
C07752=1034.474,113.929,-97.442,169.287,42.091,157.913
C07753=1034.480,114.179,-97.463,169.289,42.091,157.913
C07754=1034.486,114.428,-97.483,169.291,42.090,157.913
C07755=1034.492,114.677,-97.503,169.294,42.089,157.913
C07756=1034.498,114.926,-97.523,169.296,42.088,157.913
C07757=1034.503,115.175,-97.544,169.299,42.088,157.913
C07758=1034.509,115.424,-97.564,169.301,42.087,157.913
C07759=1034.516,115.673,-97.584,169.303,42.087,157.913
C07760=1034.522,115.922,-97.604,169.306,42.086,157.913
C07761=1034.527,116.171,-97.625,169.308,42.085,157.913
C07762=1034.534,116.421,-97.645,169.310,42.084,157.913
C07763=1034.540,116.670,-97.665,169.313,42.084,157.913
C07764=1034.546,116.919,-97.685,169.315,42.083,157.913
C07765=1034.552,117.168,-97.706,169.318,42.083,157.913
C07766=1034.558,117.417,-97.726,169.319,42.082,157.913
C07767=1034.564,117.666,-97.746,169.321,42.081,157.913
C07768=1034.570,117.916,-97.766,169.324,42.080,157.913
C07769=1034.576,118.165,-97.787,169.326,42.080,157.913
C07770=1034.582,118.413,-97.806,169.329,42.079,157.913
C07771=1034.588,118.663,-97.827,169.331,42.079,157.913
C07772=1034.594,118.911,-97.847,169.333,42.078,157.913
C07773=1034.600,119.161,-97.868,169.336,42.077,157.913
C07774=1034.606,119.410,-97.888,169.338,42.076,157.913
C07775=1034.612,119.659,-97.908,169.341,42.076,157.913
C07776=1034.619,119.908,-97.929,169.343,42.075,157.913
C07777=1034.624,120.157,-97.949,169.345,42.075,157.913
C07778=1034.631,120.407,-97.970,169.348,42.074,157.913
C07779=1034.637,120.655,-97.990,169.350,42.073,157.913
C07780=1034.643,120.904,-98.010,169.353,42.072,157.913
C07781=1034.649,121.154,-98.031,169.355,42.072,157.913
C07782=1034.655,121.402,-98.051,169.356,42.071,157.913
C07783=1034.662,121.652,-98.071,169.360,42.071,157.913
C07784=1034.668,121.901,-98.091,169.361,42.070,157.913
C07785=1034.674,122.150,-98.113,169.364,42.069,157.913
C07786=1034.680,122.399,-98.133,169.366,42.068,157.913
C07787=1034.686,122.648,-98.153,169.369,42.068,157.913
C07788=1034.692,122.897,-98.173,169.371,42.067,157.913
C07789=1034.698,123.146,-98.195,169.374,42.066,157.913
C07790=1034.704,123.395,-98.215,169.376,42.066,157.913
C07791=1034.710,123.644,-98.235,169.378,42.065,157.913
C07792=1034.716,123.894,-98.256,169.381,42.064,157.913
C07793=1034.723,124.142,-98.276,169.383,42.063,157.913
C07794=1034.730,124.429,-98.300,169.386,42.063,157.913
C07795=1034.737,124.714,-98.323,169.389,42.062,157.913
C07796=1034.744,124.999,-98.347,169.392,42.061,157.914
C07797=1034.752,125.285,-98.370,169.395,42.060,157.914
C07798=1034.757,125.534,-98.391,169.396,42.059,157.913
C07799=1034.764,125.783,-98.412,169.398,42.059,157.914
C07800=1034.770,126.031,-98.432,169.401,42.058,157.913
C07801=1034.776,126.281,-98.452,169.403,42.058,157.914
C07802=1034.782,126.529,-98.473,169.406,42.056,157.914
C07803=1034.789,126.779,-98.493,169.408,42.056,157.914
C07804=1034.795,127.028,-98.513,169.411,42.055,157.914
C07805=1034.801,127.277,-98.535,169.413,42.055,157.914
C07806=1034.807,127.526,-98.555,169.416,42.054,157.914
C07807=1034.813,127.775,-98.575,169.418,42.053,157.914
C07808=1034.819,128.024,-98.597,169.421,42.052,157.914
C07809=1034.825,128.273,-98.617,169.423,42.051,157.914
C07810=1034.832,128.522,-98.638,169.426,42.051,157.914
C07811=1034.838,128.771,-98.659,169.428,42.050,157.914
C07812=1034.844,129.021,-98.679,169.431,42.050,157.914
C07813=1034.851,129.270,-98.700,169.432,42.049,157.914
C07814=1034.857,129.518,-98.720,169.435,42.048,157.914
C07815=1034.863,129.768,-98.742,169.437,42.047,157.914
C07816=1034.869,130.016,-98.761,169.440,42.046,157.914
C07817=1034.876,130.265,-98.783,169.442,42.046,157.914
C07818=1034.882,130.515,-98.803,169.445,42.045,157.914
C07819=1034.888,130.763,-98.824,169.447,42.045,157.914
C07820=1034.894,131.013,-98.845,169.450,42.043,157.914
C07821=1034.901,131.262,-98.866,169.452,42.043,157.914
C07822=1034.906,131.511,-98.887,169.454,42.043,157.914
C07823=1034.912,131.760,-98.908,169.457,42.042,157.914
C07824=1034.918,132.009,-98.928,169.459,42.042,157.914
C07825=1034.925,132.258,-98.950,169.462,42.040,157.914
C07826=1034.931,132.507,-98.971,169.464,42.040,157.914
C07827=1034.937,132.757,-98.991,169.467,42.040,157.914
C07828=1034.943,133.006,-99.013,169.469,42.039,157.914
C07829=1034.949,133.255,-99.033,169.472,42.038,157.914
C07830=1034.955,133.504,-99.055,169.473,42.037,157.914
C07831=1034.961,133.752,-99.076,169.477,42.037,157.914
C07832=1034.967,134.002,-99.096,169.479,42.037,157.914
C07833=1034.973,134.251,-99.118,169.481,42.036,157.914
C07834=1034.980,134.499,-99.139,169.483,42.035,157.914
C07835=1034.986,134.749,-99.160,169.486,42.034,157.914
C07836=1034.992,134.998,-99.181,169.488,42.034,157.914
C07837=1034.998,135.246,-99.202,169.491,42.033,157.914
C07838=1035.004,135.496,-99.223,169.493,42.033,157.914
C07839=1035.010,135.745,-99.244,169.496,42.032,157.915
C07840=1035.016,135.994,-99.265,169.498,42.031,157.914
C07841=1035.023,136.243,-99.287,169.501,42.031,157.915
C07842=1035.028,136.493,-99.308,169.503,42.030,157.915
C07843=1035.035,136.741,-99.328,169.506,42.029,157.915
C07844=1035.041,136.990,-99.350,169.508,42.029,157.915
C07845=1035.047,137.239,-99.372,169.511,42.028,157.915
C07846=1035.053,137.487,-99.392,169.513,42.028,157.915
C07847=1035.059,137.737,-99.413,169.516,42.027,157.915
C07848=1035.065,137.986,-99.435,169.518,42.026,157.915
C07849=1035.071,138.235,-99.456,169.521,42.026,157.915
C07850=1035.078,138.484,-99.477,169.523,42.026,157.915
C07851=1035.084,138.733,-99.499,169.526,42.025,157.915
C07852=1035.089,138.982,-99.519,169.528,42.024,157.915
C07853=1035.095,139.231,-99.541,169.531,42.024,157.915
C07854=1035.102,139.480,-99.562,169.533,42.023,157.915
C07855=1035.108,139.729,-99.584,169.536,42.022,157.915
C07856=1035.114,139.978,-99.605,169.538,42.022,157.915
C07857=1035.120,140.227,-99.626,169.541,42.021,157.915
C07858=1035.127,140.512,-99.651,169.543,42.021,157.915
C07859=1035.134,140.798,-99.675,169.546,42.020,157.915
C07860=1035.141,141.083,-99.700,169.548,42.019,157.915
C07861=1035.148,141.368,-99.725,169.552,42.019,157.915
C07862=1035.154,141.617,-99.746,169.555,42.018,157.916
C07863=1035.160,141.866,-99.768,169.556,42.017,157.915
C07864=1035.166,142.115,-99.789,169.559,42.017,157.916
C07865=1035.172,142.364,-99.811,169.561,42.017,157.916
C07866=1035.178,142.614,-99.833,169.564,42.016,157.916
C07867=1035.184,142.862,-99.854,169.566,42.015,157.916
C07868=1035.190,143.111,-99.876,169.569,42.015,157.916
C07869=1035.197,143.360,-99.897,169.571,42.015,157.916
C07870=1035.203,143.609,-99.918,169.574,42.014,157.916
C07871=1035.209,143.859,-99.940,169.576,42.013,157.916
C07872=1035.215,144.107,-99.961,169.579,42.013,157.916
C07873=1035.221,144.356,-99.983,169.581,42.012,157.916
C07874=1035.227,144.605,-100.004,169.584,42.011,157.916
C07875=1035.233,144.855,-100.026,169.586,42.011,157.916
C07876=1035.239,145.103,-100.047,169.589,42.011,157.916
C07877=1035.245,145.352,-100.069,169.592,42.010,157.916
C07878=1035.251,145.602,-100.091,169.594,42.009,157.916
C07879=1035.258,145.851,-100.112,169.597,42.009,157.916
C07880=1035.264,146.100,-100.133,169.599,42.008,157.916
C07881=1035.271,146.349,-100.155,169.602,42.008,157.916
C07882=1035.276,146.597,-100.177,169.604,42.007,157.916
C07883=1035.283,146.846,-100.198,169.607,42.007,157.917
C07884=1035.289,147.095,-100.220,169.609,42.006,157.917
C07885=1035.295,147.344,-100.242,169.612,42.006,157.917
C07886=1035.300,147.594,-100.264,169.615,42.005,157.917
C07887=1035.307,147.843,-100.286,169.617,42.005,157.917
C07888=1035.312,148.091,-100.308,169.620,42.004,157.917
C07889=1035.319,148.340,-100.329,169.622,42.003,157.917
C07890=1035.325,148.589,-100.351,169.625,42.003,157.917
C07891=1035.331,148.838,-100.373,169.627,42.003,157.917
C07892=1035.337,149.087,-100.395,169.630,42.002,157.917
C07893=1035.344,149.336,-100.417,169.632,42.001,157.917
C07894=1035.350,149.586,-100.438,169.635,42.001,157.917
C07895=1035.355,149.834,-100.461,169.638,42.000,157.917
C07896=1035.361,150.083,-100.482,169.640,42.000,157.917
C07897=1035.367,150.332,-100.504,169.643,42.000,157.917
C07898=1035.374,150.581,-100.526,169.645,41.999,157.918
C07899=1035.380,150.830,-100.548,169.648,41.998,157.917
C07900=1035.386,151.079,-100.570,169.650,41.998,157.918
C07901=1035.392,151.328,-100.593,169.653,41.998,157.918
C07902=1035.398,151.577,-100.614,169.656,41.997,157.918
C07903=1035.403,151.826,-100.635,169.658,41.997,157.918
C07904=1035.410,152.074,-100.658,169.661,41.996,157.918
C07905=1035.416,152.324,-100.679,169.663,41.996,157.918
C07906=1035.422,152.572,-100.702,169.666,41.995,157.918
C07907=1035.428,152.822,-100.724,169.669,41.995,157.918
C07908=1035.434,153.071,-100.746,169.671,41.994,157.918
C07909=1035.441,153.320,-100.768,169.674,41.994,157.918
C07910=1035.447,153.569,-100.790,169.676,41.993,157.918
C07911=1035.453,153.817,-100.812,169.679,41.993,157.918
C07912=1035.459,154.067,-100.834,169.682,41.992,157.918
C07913=1035.465,154.315,-100.857,169.684,41.992,157.918
C07914=1035.471,154.565,-100.878,169.687,41.991,157.919
C07915=1035.477,154.814,-100.901,169.689,41.991,157.919
C07916=1035.483,155.062,-100.922,169.692,41.991,157.919
C07917=1035.489,155.311,-100.945,169.694,41.990,157.919
C07918=1035.494,155.560,-100.967,169.697,41.989,157.919
C07919=1035.501,155.809,-100.989,169.700,41.989,157.919
C07920=1035.507,156.058,-101.011,169.702,41.989,157.919
C07921=1035.513,156.307,-101.034,169.705,41.988,157.919
C07922=1035.521,156.592,-101.059,169.708,41.988,157.919
C07923=1035.528,156.877,-101.084,169.711,41.987,157.919
C07924=1035.534,157.162,-101.109,169.714,41.987,157.919
C07925=1035.542,157.447,-101.135,169.717,41.986,157.919
C07926=1035.547,157.696,-101.158,169.719,41.986,157.920
C07927=1035.554,157.945,-101.180,169.722,41.986,157.920
C07928=1035.560,158.194,-101.202,169.725,41.985,157.920
C07929=1035.566,158.443,-101.225,169.727,41.984,157.920
C07930=1035.572,158.692,-101.247,169.730,41.984,157.920
C07931=1035.578,158.941,-101.270,169.733,41.984,157.920
C07932=1035.584,159.190,-101.291,169.735,41.983,157.920
C07933=1035.590,159.438,-101.314,169.738,41.983,157.920
C07934=1035.596,159.687,-101.337,169.741,41.982,157.920
C07935=1035.602,159.936,-101.359,169.743,41.982,157.920
C07936=1035.608,160.185,-101.381,169.746,41.982,157.920
C07937=1035.614,160.434,-101.404,169.748,41.981,157.920
C07938=1035.620,160.683,-101.427,169.751,41.981,157.921
C07939=1035.626,160.932,-101.450,169.755,41.980,157.921
C07940=1035.632,161.181,-101.473,169.757,41.981,157.921
C07941=1035.637,161.430,-101.495,169.760,41.980,157.921
C07942=1035.643,161.679,-101.517,169.762,41.980,157.921
C07943=1035.649,161.928,-101.540,169.765,41.980,157.921
C07944=1035.655,162.177,-101.563,169.768,41.979,157.921
C07945=1035.661,162.426,-101.586,169.770,41.979,157.921
C07946=1035.667,162.674,-101.608,169.773,41.979,157.921
C07947=1035.673,162.923,-101.631,169.775,41.978,157.922
C07948=1035.679,163.172,-101.654,169.778,41.978,157.922
C07949=1035.684,163.421,-101.677,169.781,41.978,157.922
C07950=1035.691,163.669,-101.699,169.783,41.978,157.922
C07951=1035.696,163.918,-101.722,169.786,41.977,157.922
C07952=1035.702,164.167,-101.745,169.789,41.977,157.922
C07953=1035.708,164.416,-101.768,169.791,41.977,157.922
C07954=1035.714,164.665,-101.791,169.794,41.976,157.922
C07955=1035.720,164.914,-101.814,169.797,41.977,157.923
C07956=1035.726,165.162,-101.837,169.800,41.976,157.923
C07957=1035.732,165.411,-101.860,169.803,41.976,157.923
C07958=1035.738,165.661,-101.883,169.805,41.975,157.923
C07959=1035.744,165.910,-101.905,169.808,41.975,157.923
C07960=1035.750,166.158,-101.928,169.811,41.974,157.923
C07961=1035.756,166.407,-101.951,169.813,41.974,157.923
C07962=1035.762,166.656,-101.974,169.816,41.974,157.923
C07963=1035.767,166.905,-101.997,169.819,41.974,157.923
C07964=1035.774,167.154,-102.019,169.821,41.974,157.923
C07965=1035.780,167.403,-102.042,169.824,41.973,157.924
C07966=1035.785,167.652,-102.065,169.827,41.973,157.924
C07967=1035.792,167.901,-102.089,169.829,41.973,157.924
C07968=1035.797,168.150,-102.111,169.832,41.973,157.924
C07969=1035.804,168.399,-102.134,169.835,41.972,157.924
C07970=1035.810,168.647,-102.157,169.837,41.972,157.924
C07971=1035.816,168.896,-102.180,169.841,41.972,157.924
C07972=1035.821,169.145,-102.203,169.844,41.971,157.924
C07973=1035.828,169.394,-102.227,169.847,41.971,157.925
C07974=1035.834,169.643,-102.249,169.849,41.971,157.925
C07975=1035.840,169.892,-102.272,169.852,41.971,157.925
C07976=1035.846,170.141,-102.295,169.855,41.970,157.925
C07977=1035.852,170.389,-102.319,169.857,41.970,157.925
C07978=1035.857,170.638,-102.342,169.860,41.969,157.925
C07979=1035.864,170.887,-102.364,169.863,41.969,157.925
C07980=1035.870,171.136,-102.387,169.865,41.969,157.925
C07981=1035.876,171.385,-102.410,169.868,41.969,157.926
C07982=1035.882,171.633,-102.434,169.871,41.969,157.926
C07983=1035.888,171.883,-102.457,169.874,41.968,157.926
C07984=1035.894,172.132,-102.480,169.876,41.968,157.926
C07985=1035.900,172.380,-102.502,169.879,41.967,157.926
C07986=1035.907,172.664,-102.529,169.883,41.968,157.926
C07987=1035.914,172.950,-102.555,169.886,41.967,157.926
C07988=1035.921,173.234,-102.582,169.890,41.967,157.926
C07989=1035.929,173.518,-102.609,169.893,41.966,157.926
C07990=1035.934,173.767,-102.632,169.895,41.966,157.927
C07991=1035.940,174.016,-102.655,169.898,41.966,157.927
C07992=1035.946,174.266,-102.678,169.901,41.966,157.927
C07993=1035.953,174.514,-102.701,169.904,41.965,157.927
C07994=1035.959,174.762,-102.724,169.906,41.965,157.927
C07995=1035.965,175.011,-102.748,169.909,41.964,157.927
C07996=1035.971,175.260,-102.771,169.912,41.965,157.927
C07997=1035.977,175.509,-102.794,169.915,41.964,157.928
C07998=1035.983,175.758,-102.818,169.918,41.964,157.928
C07999=1035.989,176.007,-102.841,169.920,41.964,157.928
C08000=1035.996,176.256,-102.864,169.923,41.963,157.928
C08001=1036.002,176.504,-102.887,169.927,41.963,157.928
C08002=1036.008,176.754,-102.911,169.930,41.963,157.928
C08003=1036.014,177.002,-102.934,169.933,41.962,157.928
C08004=1036.021,177.251,-102.958,169.935,41.962,157.928
C08005=1036.027,177.500,-102.981,169.938,41.962,157.928
C08006=1036.032,177.749,-103.004,169.941,41.962,157.929
C08007=1036.040,177.997,-103.028,169.944,41.961,157.929
C08008=1036.045,178.246,-103.051,169.947,41.961,157.929
C08009=1036.051,178.494,-103.074,169.949,41.961,157.929
C08010=1036.058,178.744,-103.098,169.952,41.961,157.929
C08011=1036.064,178.992,-103.121,169.955,41.961,157.929
C08012=1036.070,179.242,-103.145,169.958,41.960,157.929
C08013=1036.076,179.490,-103.168,169.961,41.960,157.930
C08014=1036.083,179.739,-103.191,169.964,41.959,157.930
C08015=1036.089,179.988,-103.215,169.967,41.960,157.930
C08016=1036.095,180.237,-103.238,169.970,41.959,157.930
C08017=1036.102,180.486,-103.262,169.973,41.959,157.930
C08018=1036.107,180.735,-103.285,169.976,41.958,157.930
C08019=1036.114,180.984,-103.309,169.979,41.958,157.930
C08020=1036.120,181.232,-103.332,169.982,41.958,157.930
C08021=1036.126,181.481,-103.356,169.984,41.958,157.931
C08022=1036.132,181.730,-103.379,169.987,41.957,157.931
C08023=1036.140,181.979,-103.402,169.990,41.958,157.931
C08024=1036.146,182.227,-103.426,169.993,41.957,157.931
C08025=1036.152,182.476,-103.450,169.996,41.957,157.931
C08026=1036.158,182.725,-103.473,169.999,41.956,157.931
C08027=1036.165,182.974,-103.497,170.003,41.956,157.931
C08028=1036.171,183.222,-103.520,170.006,41.956,157.932
C08029=1036.177,183.472,-103.544,170.008,41.956,157.932
C08030=1036.182,183.721,-103.568,170.011,41.956,157.932
C08031=1036.188,183.969,-103.591,170.014,41.956,157.932
C08032=1036.194,184.218,-103.616,170.017,41.956,157.932
C08033=1036.200,184.466,-103.640,170.020,41.956,157.932
C08034=1036.207,184.715,-103.664,170.022,41.956,157.933
C08035=1036.212,184.964,-103.688,170.026,41.956,157.933
C08036=1036.219,185.213,-103.712,170.029,41.955,157.933
C08037=1036.224,185.462,-103.736,170.032,41.956,157.933
C08038=1036.230,185.710,-103.760,170.035,41.956,157.933
C08039=1036.236,185.959,-103.785,170.037,41.955,157.933
C08040=1036.242,186.207,-103.808,170.040,41.956,157.934
C08041=1036.248,186.457,-103.833,170.043,41.955,157.934
C08042=1036.254,186.705,-103.857,170.047,41.955,157.934
C08043=1036.260,186.955,-103.880,170.050,41.955,157.934
C08044=1036.266,187.203,-103.905,170.053,41.955,157.934
C08045=1036.272,187.452,-103.929,170.055,41.956,157.935
C08046=1036.278,187.700,-103.953,170.058,41.955,157.935
C08047=1036.285,187.949,-103.977,170.061,41.955,157.935
C08048=1036.290,188.198,-104.001,170.064,41.955,157.935
C08049=1036.296,188.447,-104.025,170.068,41.955,157.935
C08050=1036.303,188.731,-104.052,170.071,41.955,157.935
C08051=1036.310,189.015,-104.081,170.074,41.956,157.936
C08052=1036.316,189.299,-104.108,170.078,41.955,157.936
C08053=1036.323,189.584,-104.136,170.081,41.955,157.936
C08054=1036.329,189.832,-104.160,170.085,41.955,157.936
C08055=1036.335,190.081,-104.184,170.088,41.955,157.936
C08056=1036.341,190.330,-104.208,170.091,41.955,157.937
C08057=1036.348,190.578,-104.233,170.094,41.955,157.937
C08058=1036.354,190.827,-104.257,170.096,41.955,157.937
C08059=1036.359,191.076,-104.282,170.099,41.955,157.937
C08060=1036.366,191.325,-104.306,170.102,41.955,157.937
C08061=1036.371,191.573,-104.330,170.106,41.955,157.938
C08062=1036.378,191.822,-104.354,170.109,41.955,157.938
C08063=1036.384,192.071,-104.379,170.112,41.955,157.938
C08064=1036.390,192.319,-104.403,170.115,41.955,157.938
C08065=1036.396,192.569,-104.428,170.118,41.955,157.938
C08066=1036.402,192.817,-104.451,170.121,41.955,157.939
C08067=1036.408,193.065,-104.477,170.125,41.955,157.939
C08068=1036.415,193.314,-104.501,170.128,41.955,157.939
C08069=1036.420,193.563,-104.525,170.131,41.955,157.939
C08070=1036.427,193.812,-104.549,170.133,41.955,157.939
C08071=1036.433,194.061,-104.574,170.136,41.955,157.940
C08072=1036.439,194.309,-104.598,170.139,41.955,157.940
C08073=1036.445,194.558,-104.623,170.142,41.955,157.940
C08074=1036.452,194.807,-104.647,170.146,41.955,157.940
C08075=1036.457,195.055,-104.672,170.149,41.955,157.940
C08076=1036.464,195.304,-104.696,170.152,41.955,157.941
C08077=1036.470,195.553,-104.721,170.155,41.955,157.941
C08078=1036.477,195.802,-104.745,170.158,41.955,157.941
C08079=1036.482,196.050,-104.769,170.161,41.955,157.941
C08080=1036.489,196.299,-104.794,170.165,41.955,157.941
C08081=1036.495,196.548,-104.819,170.168,41.955,157.942
C08082=1036.501,196.796,-104.844,170.171,41.955,157.942
C08083=1036.507,197.045,-104.868,170.174,41.955,157.942
C08084=1036.513,197.294,-104.892,170.177,41.955,157.942
C08085=1036.520,197.543,-104.917,170.181,41.956,157.942
C08086=1036.526,197.792,-104.942,170.184,41.955,157.943
C08087=1036.532,198.040,-104.966,170.187,41.955,157.943
C08088=1036.538,198.289,-104.991,170.190,41.955,157.943
C08089=1036.545,198.537,-105.015,170.193,41.956,157.943
C08090=1036.551,198.787,-105.040,170.196,41.955,157.943
C08091=1036.557,199.034,-105.064,170.199,41.955,157.944
C08092=1036.563,199.283,-105.089,170.203,41.956,157.944
C08093=1036.570,199.532,-105.114,170.206,41.956,157.944
C08094=1036.576,199.781,-105.138,170.209,41.955,157.944
C08095=1036.582,200.030,-105.164,170.212,41.956,157.944
C08096=1036.589,200.279,-105.188,170.215,41.956,157.945
C08097=1036.595,200.527,-105.213,170.219,41.956,157.945
C08098=1036.601,200.776,-105.237,170.222,41.956,157.945
C08099=1036.607,201.024,-105.262,170.225,41.956,157.945
C08100=1036.614,201.273,-105.287,170.228,41.956,157.946
C08101=1036.620,201.522,-105.312,170.231,41.956,157.946
C08102=1036.626,201.771,-105.337,170.235,41.956,157.946
C08103=1036.631,202.019,-105.362,170.238,41.957,157.946
C08104=1036.638,202.268,-105.388,170.241,41.957,157.946
C08105=1036.643,202.517,-105.412,170.244,41.957,157.947
C08106=1036.650,202.765,-105.437,170.247,41.957,157.947
C08107=1036.657,203.014,-105.462,170.251,41.957,157.947
C08108=1036.663,203.263,-105.488,170.254,41.958,157.947
C08109=1036.668,203.511,-105.512,170.257,41.958,157.948
C08110=1036.674,203.760,-105.537,170.260,41.958,157.948
C08111=1036.681,204.009,-105.563,170.264,41.958,157.948
C08112=1036.687,204.257,-105.588,170.267,41.958,157.948
C08113=1036.693,204.506,-105.613,170.271,41.958,157.949
C08114=1036.719,205.556,-105.719,170.582,42.063,157.990
C08115=1036.728,205.882,-105.754,170.584,42.064,157.991
C08116=1036.737,206.208,-105.788,170.588,42.065,157.991
C08117=1036.746,206.534,-105.823,170.590,42.067,157.991
C08118=1036.754,206.859,-105.857,170.594,42.068,157.992
C08119=1036.761,207.108,-105.884,170.596,42.069,157.992
C08120=1036.768,207.356,-105.910,170.598,42.070,157.993
C08121=1036.775,207.605,-105.936,170.601,42.070,157.993
C08122=1036.781,207.854,-105.963,170.603,42.071,157.993
C08123=1036.788,208.102,-105.989,170.606,42.072,157.994
C08124=1036.795,208.350,-106.017,170.608,42.073,157.994
C08125=1036.802,208.599,-106.044,170.610,42.074,157.994
C08126=1036.808,208.847,-106.070,170.613,42.075,157.995
C08127=1036.815,209.096,-106.096,170.615,42.076,157.995
C08128=1036.822,209.344,-106.122,170.618,42.077,157.995
C08129=1036.828,209.593,-106.149,170.620,42.078,157.996
C08130=1036.835,209.841,-106.176,170.622,42.079,157.996
C08131=1036.842,210.089,-106.202,170.625,42.080,157.996
C08132=1036.848,210.338,-106.229,170.627,42.081,157.997
C08133=1036.856,210.587,-106.256,170.630,42.082,157.997
C08134=1036.861,210.835,-106.282,170.632,42.083,157.998
C08135=1036.868,211.084,-106.309,170.634,42.084,157.998
C08136=1036.876,211.332,-106.336,170.637,42.085,157.998
C08137=1036.882,211.580,-106.363,170.639,42.086,157.999
C08138=1036.889,211.829,-106.389,170.642,42.087,157.999
C08139=1036.895,212.078,-106.417,170.644,42.088,157.999
C08140=1036.902,212.326,-106.443,170.646,42.089,158.000
C08141=1036.908,212.575,-106.470,170.649,42.090,158.000
C08142=1036.916,212.823,-106.497,170.651,42.091,158.000
C08143=1036.921,213.071,-106.524,170.654,42.092,158.001
C08144=1036.929,213.320,-106.550,170.656,42.092,158.001
C08145=1036.935,213.568,-106.578,170.658,42.093,158.001
C08146=1036.942,213.817,-106.604,170.661,42.094,158.002
C08147=1036.948,214.065,-106.631,170.663,42.095,158.002
C08148=1036.955,214.314,-106.659,170.666,42.096,158.002
C08149=1036.962,214.563,-106.685,170.668,42.097,158.003
C08150=1036.968,214.810,-106.712,170.670,42.098,158.003
C08151=1036.975,215.059,-106.739,170.673,42.099,158.004
C08152=1036.982,215.308,-106.766,170.675,42.100,158.004
C08153=1036.989,215.556,-106.793,170.678,42.101,158.004
C08154=1036.995,215.805,-106.820,170.680,42.103,158.005
C08155=1037.002,216.053,-106.847,170.683,42.104,158.005
C08156=1037.008,216.302,-106.874,170.685,42.105,158.005
C08157=1037.016,216.550,-106.901,170.687,42.106,158.006
C08158=1037.022,216.798,-106.927,170.690,42.106,158.006
C08159=1037.029,217.046,-106.955,170.692,42.107,158.007
C08160=1037.035,217.296,-106.982,170.696,42.108,158.007
C08161=1037.042,217.544,-107.009,170.698,42.109,158.007
C08162=1037.049,217.792,-107.035,170.700,42.110,158.008
C08163=1037.055,218.040,-107.063,170.703,42.111,158.008
C08164=1037.062,218.289,-107.090,170.705,42.112,158.008
C08165=1037.069,218.538,-107.117,170.708,42.113,158.009
C08166=1037.076,218.786,-107.144,170.710,42.114,158.009
C08167=1037.082,219.034,-107.171,170.712,42.115,158.009
C08168=1037.089,219.283,-107.197,170.715,42.116,158.010
C08169=1037.096,219.531,-107.225,170.717,42.117,158.010
C08170=1037.103,219.780,-107.253,170.721,42.118,158.011
C08171=1037.112,220.111,-107.288,170.723,42.119,158.011
C08172=1037.121,220.443,-107.325,170.727,42.121,158.012
C08173=1037.129,220.774,-107.361,170.730,42.121,158.012
C08174=1037.138,221.105,-107.398,170.734,42.123,158.012
C08175=1037.145,221.354,-107.426,170.736,42.124,158.013
C08176=1037.151,221.602,-107.452,170.739,42.125,158.013
C08177=1037.158,221.850,-107.480,170.741,42.126,158.014
C08178=1037.165,222.099,-107.508,170.744,42.127,158.014
C08179=1037.171,222.347,-107.535,170.746,42.128,158.014
C08180=1037.178,222.596,-107.562,170.748,42.129,158.015
C08181=1037.185,222.844,-107.589,170.751,42.130,158.015
C08182=1037.192,223.093,-107.617,170.754,42.131,158.016
C08183=1037.198,223.341,-107.645,170.757,42.132,158.016
C08184=1037.205,223.589,-107.672,170.759,42.133,158.016
C08185=1037.211,223.838,-107.699,170.762,42.134,158.017
C08186=1037.218,224.087,-107.727,170.764,42.135,158.017
C08187=1037.225,224.335,-107.754,170.766,42.136,158.017
C08188=1037.232,224.583,-107.782,170.769,42.137,158.018
C08189=1037.238,224.832,-107.810,170.772,42.138,158.018
C08190=1037.245,225.080,-107.837,170.775,42.139,158.019
C08191=1037.251,225.328,-107.865,170.777,42.140,158.019
C08192=1037.258,225.577,-107.892,170.780,42.141,158.019
C08193=1037.264,225.825,-107.919,170.782,42.142,158.020
C08194=1037.272,226.073,-107.947,170.785,42.143,158.020
C08195=1037.278,226.322,-107.974,170.787,42.144,158.020
C08196=1037.285,226.570,-108.002,170.790,42.145,158.021
C08197=1037.292,226.819,-108.030,170.793,42.146,158.021
C08198=1037.298,227.067,-108.057,170.795,42.147,158.022
C08199=1037.305,227.316,-108.085,170.798,42.148,158.022
C08200=1037.312,227.564,-108.112,170.800,42.149,158.022
C08201=1037.319,227.812,-108.140,170.803,42.150,158.023
C08202=1037.326,228.061,-108.168,170.806,42.151,158.023
C08203=1037.332,228.309,-108.196,170.808,42.152,158.024
C08204=1037.339,228.558,-108.223,170.811,42.153,158.024
C08205=1037.346,228.806,-108.251,170.813,42.154,158.024
C08206=1037.353,229.054,-108.279,170.817,42.155,158.025
C08207=1037.359,229.303,-108.306,170.819,42.156,158.025
C08208=1037.365,229.552,-108.335,170.822,42.157,158.026
C08209=1037.372,229.800,-108.363,170.824,42.158,158.026
C08210=1037.378,230.048,-108.390,170.826,42.159,158.026
C08211=1037.385,230.296,-108.418,170.830,42.160,158.027
C08212=1037.392,230.544,-108.446,170.832,42.161,158.027
C08213=1037.398,230.792,-108.474,170.835,42.163,158.028
C08214=1037.405,231.041,-108.502,170.837,42.164,158.028
C08215=1037.412,231.289,-108.529,170.840,42.165,158.028
C08216=1037.418,231.538,-108.557,170.843,42.165,158.029
C08217=1037.425,231.786,-108.585,170.845,42.166,158.029
C08218=1037.431,232.034,-108.614,170.848,42.168,158.029
C08219=1037.438,232.283,-108.641,170.850,42.169,158.030
C08220=1037.445,232.531,-108.669,170.853,42.170,158.030
C08221=1037.451,232.780,-108.697,170.856,42.171,158.031
C08222=1037.458,233.028,-108.725,170.859,42.172,158.031
C08223=1037.464,233.276,-108.754,170.861,42.173,158.031
C08224=1037.471,233.525,-108.781,170.864,42.174,158.032
C08225=1037.478,233.773,-108.810,170.867,42.175,158.032
C08226=1037.485,234.022,-108.838,170.870,42.176,158.033
C08227=1037.494,234.345,-108.875,170.873,42.178,158.033
C08228=1037.502,234.670,-108.911,170.877,42.179,158.034
C08229=1037.511,234.993,-108.948,170.880,42.180,158.034
C08230=1037.519,235.317,-108.985,170.884,42.181,158.035
C08231=1037.526,235.565,-109.013,170.887,42.183,158.035
C08232=1037.532,235.814,-109.041,170.889,42.184,158.036
C08233=1037.539,236.062,-109.069,170.891,42.185,158.036
C08234=1037.546,236.310,-109.097,170.895,42.186,158.036
C08235=1037.553,236.559,-109.126,170.897,42.187,158.037
C08236=1037.559,236.807,-109.154,170.900,42.188,158.037
C08237=1037.566,237.056,-109.182,170.902,42.189,158.038
C08238=1037.573,237.304,-109.210,170.906,42.190,158.038
C08239=1037.579,237.552,-109.238,170.908,42.191,158.038
C08240=1037.586,237.800,-109.267,170.911,42.192,158.039
C08241=1037.592,238.049,-109.295,170.914,42.193,158.039
C08242=1037.599,238.296,-109.323,170.917,42.195,158.040
C08243=1037.606,238.546,-109.352,170.919,42.196,158.040
C08244=1037.613,238.794,-109.380,170.922,42.196,158.040
C08245=1037.620,239.042,-109.408,170.925,42.197,158.041
C08246=1037.626,239.290,-109.437,170.927,42.199,158.041
C08247=1037.633,239.538,-109.466,170.930,42.200,158.042
C08248=1037.640,239.787,-109.493,170.933,42.201,158.042
C08249=1037.646,240.035,-109.522,170.936,42.202,158.043
C08250=1037.653,240.284,-109.551,170.938,42.203,158.043
C08251=1037.660,240.532,-109.579,170.942,42.204,158.043
C08252=1037.667,240.780,-109.607,170.944,42.205,158.044
C08253=1037.673,241.028,-109.636,170.947,42.206,158.044
C08254=1037.679,241.276,-109.665,170.950,42.207,158.045
C08255=1037.686,241.524,-109.693,170.953,42.209,158.045
C08256=1037.693,241.774,-109.722,170.955,42.210,158.045
C08257=1037.700,242.021,-109.750,170.959,42.211,158.046
C08258=1037.706,242.270,-109.779,170.961,42.212,158.046
C08259=1037.713,242.518,-109.807,170.964,42.213,158.047
C08260=1037.719,242.766,-109.836,170.967,42.214,158.047
C08261=1037.726,243.015,-109.866,170.970,42.215,158.048
C08262=1037.733,243.263,-109.894,170.972,42.216,158.048
C08263=1037.739,243.511,-109.923,170.976,42.218,158.049
C08264=1037.746,243.759,-109.951,170.978,42.219,158.049
C08265=1037.752,244.008,-109.980,170.980,42.220,158.049
C08266=1037.760,244.256,-110.009,170.984,42.221,158.050
C08267=1037.766,244.504,-110.038,170.986,42.222,158.050
C08268=1037.772,244.752,-110.067,170.990,42.223,158.051
C08269=1037.779,245.001,-110.094,170.992,42.224,158.051
C08270=1037.785,245.249,-110.124,170.995,42.226,158.052
C08271=1037.792,245.498,-110.153,170.998,42.227,158.052
C08272=1037.798,245.746,-110.182,171.001,42.228,158.052
C08273=1037.805,245.994,-110.210,171.004,42.229,158.053
C08274=1037.811,246.242,-110.239,171.007,42.230,158.053
C08275=1037.818,246.491,-110.269,171.010,42.231,158.054
C08276=1037.824,246.739,-110.298,171.012,42.233,158.054
C08277=1037.831,246.987,-110.327,171.016,42.234,158.055
C08278=1037.837,247.235,-110.356,171.018,42.235,158.055
C08279=1037.843,247.483,-110.385,171.021,42.236,158.055
C08280=1037.851,247.732,-110.414,171.024,42.238,158.056
C08281=1037.857,247.980,-110.443,171.027,42.239,158.056
C08282=1037.863,248.228,-110.472,171.030,42.240,158.057
C08283=1037.872,248.546,-110.509,171.034,42.241,158.057
C08284=1037.880,248.864,-110.547,171.037,42.243,158.058
C08285=1037.889,249.181,-110.584,171.041,42.244,158.059
C08286=1037.897,249.501,-110.622,171.045,42.246,158.059
C08287=1037.904,249.748,-110.651,171.047,42.247,158.060
C08288=1037.911,249.996,-110.680,171.051,42.249,158.060
C08289=1037.917,250.244,-110.709,171.053,42.249,158.060
C08290=1037.924,250.493,-110.738,171.056,42.251,158.061
C08291=1037.930,250.741,-110.767,171.059,42.252,158.061
C08292=1037.937,250.990,-110.797,171.062,42.253,158.062
C08293=1037.943,251.237,-110.827,171.065,42.254,158.062
C08294=1037.950,251.485,-110.855,171.068,42.256,158.063
C08295=1037.957,251.734,-110.884,171.071,42.256,158.063
C08296=1037.963,251.982,-110.914,171.074,42.258,158.064
C08297=1037.970,252.230,-110.943,171.077,42.259,158.064
C08298=1037.977,252.479,-110.973,171.080,42.260,158.065
C08299=1037.983,252.727,-111.002,171.083,42.262,158.065
C08300=1037.989,252.975,-111.031,171.086,42.263,158.066
C08301=1037.996,253.223,-111.061,171.089,42.264,158.066
C08302=1038.003,253.471,-111.089,171.092,42.265,158.066
C08303=1038.010,253.720,-111.119,171.095,42.267,158.067
C08304=1038.017,253.968,-111.148,171.098,42.267,158.067
C08305=1038.024,254.216,-111.178,171.101,42.269,158.068
C08306=1038.030,254.464,-111.207,171.104,42.270,158.068
C08307=1038.036,254.712,-111.236,171.107,42.271,158.069
C08308=1038.043,254.960,-111.266,171.110,42.272,158.069
C08309=1038.050,255.209,-111.295,171.113,42.273,158.070
C08310=1038.058,255.457,-111.325,171.116,42.274,158.070
C08311=1038.064,255.705,-111.354,171.119,42.276,158.071
C08312=1038.071,255.953,-111.383,171.122,42.277,158.071
C08313=1038.077,256.201,-111.413,171.125,42.278,158.071
C08314=1038.084,256.450,-111.442,171.128,42.280,158.072
C08315=1038.091,256.697,-111.472,171.131,42.280,158.072
C08316=1038.097,256.946,-111.501,171.134,42.282,158.073
C08317=1038.104,257.194,-111.531,171.137,42.283,158.073
C08318=1038.111,257.443,-111.561,171.140,42.284,158.074
C08319=1038.117,257.690,-111.590,171.143,42.285,158.074
C08320=1038.125,257.939,-111.619,171.146,42.286,158.075
C08321=1038.132,258.186,-111.649,171.149,42.288,158.075
C08322=1038.138,258.435,-111.678,171.153,42.289,158.076
C08323=1038.145,258.682,-111.708,171.156,42.290,158.076
C08324=1038.152,258.931,-111.737,171.159,42.291,158.077
C08325=1038.159,259.179,-111.768,171.162,42.292,158.077
C08326=1038.165,259.428,-111.797,171.165,42.293,158.077
C08327=1038.172,259.676,-111.827,171.168,42.295,158.078
C08328=1038.179,259.924,-111.856,171.171,42.296,158.078
C08329=1038.186,260.172,-111.886,171.174,42.297,158.079
C08330=1038.192,260.420,-111.916,171.178,42.298,158.079
C08331=1038.200,260.668,-111.945,171.180,42.299,158.080
C08332=1038.207,260.916,-111.975,171.184,42.301,158.080
C08333=1038.214,261.164,-112.004,171.186,42.302,158.081
C08334=1038.220,261.413,-112.034,171.190,42.303,158.081
C08335=1038.228,261.661,-112.064,171.194,42.304,158.082
C08336=1038.234,261.908,-112.094,171.196,42.305,158.082
C08337=1038.240,262.158,-112.124,171.200,42.307,158.083
C08338=1038.247,262.405,-112.153,171.202,42.308,158.083
C08339=1038.256,262.722,-112.192,171.207,42.310,158.084
C08340=1038.264,263.038,-112.230,171.211,42.312,158.084
C08341=1038.273,263.355,-112.268,171.214,42.313,158.085
C08342=1038.281,263.671,-112.307,171.218,42.315,158.086
C08343=1038.288,263.919,-112.337,171.222,42.316,158.086
C08344=1038.294,264.168,-112.366,171.225,42.318,158.087
C08345=1038.301,264.416,-112.397,171.228,42.319,158.087
C08346=1038.308,264.664,-112.427,171.231,42.320,158.088
C08347=1038.315,264.912,-112.457,171.234,42.322,158.088
C08348=1038.321,265.160,-112.488,171.238,42.323,158.089
C08349=1038.328,265.409,-112.518,171.241,42.324,158.089
C08350=1038.335,265.656,-112.548,171.244,42.325,158.090
C08351=1038.341,265.905,-112.578,171.247,42.327,158.090
C08352=1038.348,266.153,-112.608,171.250,42.328,158.091
C08353=1038.355,266.400,-112.638,171.253,42.330,158.091
C08354=1038.362,266.649,-112.668,171.257,42.330,158.092
C08355=1038.368,266.897,-112.699,171.259,42.332,158.092
C08356=1038.375,267.145,-112.729,171.263,42.333,158.093
C08357=1038.381,267.393,-112.759,171.267,42.335,158.093
C08358=1038.388,267.641,-112.790,171.269,42.336,158.094
C08359=1038.395,267.889,-112.819,171.273,42.337,158.094
C08360=1038.402,268.137,-112.851,171.276,42.338,158.095
C08361=1038.409,268.385,-112.881,171.279,42.340,158.095
C08362=1038.415,268.633,-112.911,171.283,42.341,158.096
C08363=1038.422,268.881,-112.941,171.285,42.343,158.096
C08364=1038.428,269.130,-112.972,171.289,42.344,158.097
C08365=1038.435,269.378,-113.002,171.292,42.345,158.097
C08366=1038.442,269.625,-113.033,171.295,42.347,158.098
C08367=1038.449,269.873,-113.063,171.299,42.348,158.098
C08368=1038.455,270.122,-113.094,171.302,42.349,158.099
C08369=1038.462,270.370,-113.124,171.305,42.351,158.099
C08370=1038.468,270.617,-113.155,171.308,42.352,158.100
C08371=1038.476,270.865,-113.185,171.312,42.353,158.100
C08372=1038.482,271.114,-113.216,171.316,42.355,158.101
C08373=1038.489,271.362,-113.246,171.318,42.356,158.101
C08374=1038.495,271.609,-113.277,171.322,42.358,158.102
C08375=1038.502,271.857,-113.307,171.325,42.359,158.103
C08376=1038.509,272.105,-113.339,171.328,42.361,158.103
C08377=1038.516,272.354,-113.370,171.332,42.362,158.104
C08378=1038.523,272.602,-113.400,171.335,42.363,158.104
C08379=1038.529,272.849,-113.431,171.338,42.365,158.105
C08380=1038.535,273.098,-113.461,171.342,42.366,158.105
C08381=1038.543,273.345,-113.492,171.345,42.368,158.106
C08382=1038.549,273.594,-113.523,171.348,42.369,158.106
C08383=1038.556,273.842,-113.553,171.351,42.371,158.107
C08384=1038.562,274.089,-113.584,171.355,42.372,158.107
C08385=1038.569,274.338,-113.615,171.359,42.373,158.108
C08386=1038.576,274.585,-113.646,171.361,42.375,158.108
C08387=1038.583,274.834,-113.676,171.365,42.376,158.109
C08388=1038.589,275.082,-113.708,171.368,42.378,158.110
C08389=1038.596,275.330,-113.739,171.372,42.379,158.110
C08390=1038.603,275.577,-113.769,171.375,42.380,158.111
C08391=1038.609,275.825,-113.801,171.378,42.382,158.111
C08392=1038.616,276.074,-113.831,171.382,42.383,158.112
C08393=1038.623,276.322,-113.863,171.385,42.385,158.112
C08394=1038.630,276.569,-113.894,171.388,42.386,158.113
C08395=1038.638,276.891,-113.933,171.393,42.388,158.113
C08396=1038.647,277.212,-113.973,171.397,42.390,158.114
C08397=1038.656,277.534,-114.014,171.402,42.392,158.115
C08398=1038.664,277.854,-114.054,171.407,42.393,158.116
C08399=1038.672,278.102,-114.085,171.409,42.395,158.116
C08400=1038.678,278.350,-114.116,171.413,42.397,158.117
C08401=1038.685,278.598,-114.147,171.417,42.398,158.117
C08402=1038.692,278.846,-114.179,171.420,42.400,158.118
C08403=1038.698,279.094,-114.210,171.423,42.401,158.118
C08404=1038.705,279.342,-114.241,171.426,42.403,158.119
C08405=1038.712,279.590,-114.273,171.430,42.404,158.120
C08406=1038.718,279.838,-114.304,171.434,42.406,158.120
C08407=1038.725,280.086,-114.335,171.438,42.407,158.121
C08408=1038.732,280.334,-114.366,171.440,42.409,158.121
C08409=1038.738,280.581,-114.397,171.444,42.410,158.122
C08410=1038.744,280.829,-114.429,171.448,42.412,158.123
C08411=1038.751,281.077,-114.460,171.451,42.414,158.123
C08412=1038.758,281.325,-114.492,171.455,42.415,158.124
C08413=1038.765,281.573,-114.523,171.457,42.416,158.124
C08414=1038.772,281.821,-114.554,171.461,42.418,158.125
C08415=1038.779,282.069,-114.585,171.465,42.420,158.125
C08416=1038.786,282.316,-114.617,171.469,42.421,158.126
C08417=1038.792,282.564,-114.648,171.472,42.422,158.127
C08418=1038.799,282.812,-114.680,171.475,42.425,158.127
C08419=1038.806,283.060,-114.711,171.479,42.426,158.128
C08420=1038.812,283.308,-114.743,171.482,42.427,158.128
C08421=1038.819,283.556,-114.774,171.486,42.429,158.129
C08422=1038.827,283.805,-114.806,171.490,42.431,158.130
C08423=1038.833,284.052,-114.837,171.493,42.432,158.130
C08424=1038.840,284.300,-114.869,171.497,42.433,158.131
C08425=1038.847,284.548,-114.900,171.500,42.435,158.131
C08426=1038.853,284.796,-114.932,171.503,42.437,158.132
C08427=1038.860,285.044,-114.963,171.507,42.438,158.132
C08428=1038.867,285.291,-114.995,171.511,42.440,158.133
C08429=1038.874,285.539,-115.027,171.515,42.442,158.134
C08430=1038.881,285.787,-115.058,171.518,42.443,158.134
C08431=1038.887,286.035,-115.089,171.522,42.444,158.135
C08432=1038.895,286.284,-115.121,171.526,42.446,158.135
C08433=1038.901,286.532,-115.153,171.528,42.448,158.136
C08434=1038.908,286.779,-115.185,171.532,42.449,158.137
C08435=1038.914,287.027,-115.217,171.536,42.451,158.137
C08436=1038.921,287.275,-115.248,171.539,42.452,158.138
C08437=1038.928,287.522,-115.280,171.543,42.454,158.138
C08438=1038.935,287.770,-115.312,171.547,42.456,158.139
C08439=1038.942,288.018,-115.343,171.550,42.457,158.140
C08440=1038.949,288.266,-115.376,171.554,42.459,158.140
C08441=1038.955,288.514,-115.408,171.558,42.460,158.141
C08442=1038.962,288.762,-115.439,171.562,42.462,158.142
C08443=1038.969,289.009,-115.471,171.564,42.464,158.142
C08444=1038.975,289.258,-115.503,171.568,42.466,158.143
C08445=1038.982,289.505,-115.536,171.572,42.467,158.143
C08446=1038.989,289.754,-115.567,171.576,42.469,158.144
C08447=1038.996,290.001,-115.600,171.579,42.470,158.145
C08448=1039.002,290.249,-115.632,171.583,42.472,158.145
C08449=1039.009,290.496,-115.664,171.587,42.474,158.146
C08450=1039.016,290.744,-115.695,171.591,42.476,158.147
C08451=1039.026,291.078,-115.739,171.595,42.478,158.147
C08452=1039.035,291.410,-115.782,171.600,42.480,158.148
C08453=1039.044,291.744,-115.825,171.605,42.482,158.149
C08454=1039.053,292.077,-115.869,171.610,42.485,158.150
C08455=1039.060,292.324,-115.901,171.614,42.486,158.150
C08456=1039.066,292.572,-115.932,171.618,42.488,158.151
C08457=1039.073,292.820,-115.965,171.622,42.489,158.152
C08458=1039.080,293.068,-115.997,171.625,42.491,158.152
C08459=1039.087,293.316,-116.029,171.629,42.493,158.153
C08460=1039.094,293.564,-116.062,171.633,42.495,158.154
C08461=1039.101,293.811,-116.094,171.637,42.497,158.154
C08462=1039.108,294.059,-116.126,171.640,42.498,158.155
C08463=1039.114,294.307,-116.158,171.644,42.500,158.156
C08464=1039.122,294.555,-116.191,171.648,42.502,158.156
C08465=1039.128,294.802,-116.224,171.652,42.503,158.157
C08466=1039.135,295.050,-116.256,171.655,42.505,158.158
C08467=1039.141,295.298,-116.288,171.659,42.507,158.158
C08468=1039.149,295.546,-116.320,171.663,42.508,158.159
C08469=1039.155,295.793,-116.353,171.667,42.510,158.160
C08470=1039.162,296.042,-116.386,171.671,42.512,158.160
C08471=1039.168,296.289,-116.419,171.674,42.514,158.161
C08472=1039.175,296.536,-116.451,171.678,42.516,158.162
C08473=1039.181,296.784,-116.484,171.682,42.518,158.162
C08474=1039.188,297.032,-116.517,171.686,42.520,158.163
C08475=1039.194,297.280,-116.550,171.690,42.522,158.164
C08476=1039.202,297.527,-116.582,171.693,42.523,158.164
C08477=1039.208,297.776,-116.615,171.697,42.525,158.165
C08478=1039.215,298.023,-116.648,171.701,42.527,158.166
C08479=1039.221,298.270,-116.681,171.705,42.529,158.166
C08480=1039.228,298.518,-116.714,171.709,42.531,158.167
C08481=1039.235,298.766,-116.746,171.712,42.533,158.168
C08482=1039.242,299.014,-116.779,171.716,42.535,158.168
C08483=1039.248,299.262,-116.812,171.720,42.536,158.169
C08484=1039.255,299.509,-116.845,171.724,42.538,158.170
C08485=1039.262,299.757,-116.877,171.728,42.540,158.171
C08486=1039.269,300.004,-116.911,171.732,42.542,158.171
C08487=1039.276,300.252,-116.944,171.735,42.544,158.172
C08488=1039.282,300.500,-116.977,171.739,42.546,158.172
C08489=1039.288,300.748,-117.009,171.743,42.548,158.173
C08490=1039.296,300.996,-117.042,171.747,42.549,158.174
C08491=1039.303,301.243,-117.075,171.751,42.551,158.175
C08492=1039.310,301.491,-117.109,171.754,42.553,158.175
C08493=1039.316,301.738,-117.141,171.759,42.555,158.176
C08494=1039.324,301.986,-117.174,171.763,42.557,158.177
C08495=1039.330,302.233,-117.207,171.767,42.559,158.177
C08496=1039.337,302.482,-117.240,171.771,42.561,158.178
C08497=1039.344,302.729,-117.274,171.775,42.563,158.179
C08498=1039.350,302.977,-117.307,171.779,42.565,158.180
C08499=1039.357,303.224,-117.339,171.782,42.567,158.180
C08500=1039.365,303.472,-117.373,171.786,42.569,158.181
C08501=1039.371,303.720,-117.406,171.790,42.571,158.182
C08502=1039.378,303.967,-117.439,171.795,42.572,158.182
C08503=1039.384,304.215,-117.472,171.799,42.574,158.183
C08504=1039.392,304.462,-117.505,171.803,42.576,158.184
C08505=1039.399,304.710,-117.539,171.806,42.578,158.185
C08506=1039.406,304.958,-117.571,171.810,42.580,158.185
C08507=1039.416,305.307,-117.619,171.817,42.583,158.186
C08508=1039.426,305.657,-117.666,171.822,42.585,158.187
C08509=1039.435,306.007,-117.712,171.828,42.588,158.188
C08510=1039.445,306.357,-117.759,171.833,42.591,158.189
C08511=1039.452,306.604,-117.793,171.837,42.593,158.190
C08512=1039.459,306.853,-117.826,171.842,42.595,158.191
C08513=1039.466,307.099,-117.859,171.846,42.597,158.192
C08514=1039.473,307.347,-117.893,171.850,42.599,158.192
C08515=1039.480,307.595,-117.926,171.853,42.601,158.193
C08516=1039.487,307.842,-117.959,171.857,42.603,158.194
C08517=1039.495,308.090,-117.993,171.862,42.605,158.195
C08518=1039.501,308.338,-118.026,171.866,42.607,158.195
C08519=1039.508,308.585,-118.060,171.870,42.609,158.196
C08520=1039.515,308.833,-118.093,171.874,42.611,158.197
C08521=1039.522,309.080,-118.127,171.879,42.612,158.197
C08522=1039.529,309.329,-118.160,171.882,42.614,158.198
C08523=1039.537,309.575,-118.193,171.886,42.616,158.199
C08524=1039.544,309.823,-118.227,171.890,42.619,158.200
C08525=1039.551,310.071,-118.261,171.895,42.621,158.200
C08526=1039.558,310.319,-118.294,171.899,42.623,158.201
C08527=1039.565,310.567,-118.328,171.903,42.624,158.202
C08528=1039.572,310.814,-118.361,171.907,42.626,158.203
C08529=1039.579,311.061,-118.395,171.912,42.629,158.203
C08530=1039.587,311.309,-118.428,171.916,42.631,158.204
C08531=1039.594,311.556,-118.462,171.920,42.633,158.205
C08532=1039.601,311.804,-118.496,171.924,42.634,158.206
C08533=1039.609,312.052,-118.530,171.928,42.636,158.206
C08534=1039.615,312.299,-118.563,171.932,42.639,158.207
C08535=1039.622,312.547,-118.598,171.936,42.641,158.208
C08536=1039.629,312.794,-118.632,171.941,42.643,158.209
C08537=1039.635,313.042,-118.666,171.945,42.645,158.210
C08538=1039.642,313.289,-118.699,171.949,42.648,158.210
C08539=1039.648,313.537,-118.734,171.953,42.649,158.211
C08540=1039.656,313.784,-118.768,171.958,42.652,158.212
C08541=1039.663,314.032,-118.802,171.962,42.654,158.213
C08542=1039.669,314.280,-118.837,171.966,42.656,158.214
C08543=1039.676,314.527,-118.870,171.970,42.659,158.214
C08544=1039.683,314.774,-118.905,171.975,42.661,158.215
C08545=1039.690,315.022,-118.939,171.979,42.663,158.216
C08546=1039.696,315.270,-118.973,171.983,42.665,158.217
C08547=1039.704,315.517,-119.008,171.987,42.668,158.218
C08548=1039.710,315.765,-119.042,171.992,42.670,158.219
C08549=1039.718,316.013,-119.076,171.996,42.672,158.219
C08550=1039.724,316.259,-119.111,172.000,42.674,158.220
C08551=1039.731,316.507,-119.145,172.005,42.676,158.221
C08552=1039.738,316.755,-119.179,172.009,42.679,158.222
C08553=1039.745,317.002,-119.214,172.013,42.681,158.223
C08554=1039.752,317.250,-119.248,172.018,42.683,158.223
C08555=1039.759,317.497,-119.283,172.022,42.685,158.224
C08556=1039.766,317.745,-119.317,172.026,42.688,158.225
C08557=1039.773,317.992,-119.352,172.031,42.690,158.226
C08558=1039.780,318.240,-119.386,172.035,42.692,158.227
C08559=1039.787,318.487,-119.421,172.039,42.695,158.228
C08560=1039.794,318.735,-119.455,172.044,42.696,158.228
C08561=1039.801,318.982,-119.490,172.048,42.699,158.229
C08562=1039.808,319.230,-119.523,172.053,42.701,158.230
C08563=1039.818,319.584,-119.573,172.058,42.705,158.231
C08564=1039.828,319.939,-119.622,172.065,42.708,158.232
C08565=1039.838,320.293,-119.672,172.071,42.711,158.234
C08566=1039.848,320.648,-119.722,172.078,42.714,158.235
C08567=1039.856,320.895,-119.756,172.082,42.717,158.236
C08568=1039.862,321.143,-119.791,172.087,42.719,158.237
C08569=1039.870,321.390,-119.826,172.091,42.721,158.237
C08570=1039.876,321.638,-119.860,172.096,42.723,158.238
C08571=1039.884,321.886,-119.896,172.100,42.726,158.239
C08572=1039.891,322.133,-119.930,172.105,42.728,158.240
C08573=1039.898,322.380,-119.965,172.109,42.731,158.241
C08574=1039.905,322.628,-119.999,172.113,42.733,158.242
C08575=1039.912,322.875,-120.034,172.118,42.735,158.243
C08576=1039.919,323.122,-120.069,172.122,42.737,158.243
C08577=1039.927,323.370,-120.104,172.127,42.740,158.244
C08578=1039.934,323.617,-120.139,172.131,42.742,158.245
C08579=1039.941,323.865,-120.173,172.136,42.745,158.246
C08580=1039.948,324.112,-120.208,172.140,42.747,158.247
C08581=1039.955,324.360,-120.243,172.145,42.749,158.248
C08582=1039.963,324.607,-120.278,172.149,42.752,158.249
C08583=1039.970,324.855,-120.313,172.154,42.754,158.249
C08584=1039.977,325.102,-120.347,172.158,42.756,158.250
C08585=1039.985,325.350,-120.383,172.163,42.759,158.251
C08586=1039.992,325.597,-120.418,172.167,42.761,158.252
C08587=1039.999,325.844,-120.453,172.172,42.763,158.253
C08588=1040.006,326.092,-120.488,172.176,42.766,158.254
C08589=1040.014,326.339,-120.523,172.182,42.768,158.255
C08590=1040.021,326.587,-120.558,172.186,42.771,158.256
C08591=1040.028,326.834,-120.592,172.191,42.773,158.257
C08592=1040.036,327.082,-120.628,172.195,42.775,158.257
C08593=1040.043,327.329,-120.662,172.200,42.778,158.258
C08594=1040.050,327.577,-120.698,172.205,42.780,158.259
C08595=1040.058,327.824,-120.734,172.209,42.783,158.260
C08596=1040.065,328.071,-120.768,172.214,42.786,158.261
C08597=1040.072,328.319,-120.804,172.218,42.788,158.262
C08598=1040.080,328.566,-120.838,172.223,42.790,158.263
C08599=1040.087,328.814,-120.874,172.228,42.793,158.264
C08600=1040.094,329.061,-120.910,172.233,42.795,158.265
C08601=1040.101,329.308,-120.945,172.237,42.798,158.266
C08602=1040.109,329.556,-120.980,172.242,42.801,158.267
C08603=1040.116,329.803,-121.016,172.247,42.803,158.268
C08604=1040.123,330.051,-121.052,172.251,42.805,158.269
C08605=1040.130,330.298,-121.088,172.256,42.808,158.270
C08606=1040.137,330.545,-121.123,172.260,42.811,158.270
C08607=1040.144,330.793,-121.158,172.266,42.813,158.271
C08608=1040.151,331.040,-121.194,172.270,42.816,158.272
C08609=1040.159,331.288,-121.230,172.275,42.818,158.273
C08610=1040.166,331.535,-121.265,172.280,42.821,158.274
C08611=1040.173,331.782,-121.302,172.284,42.824,158.275
C08612=1040.180,332.030,-121.337,172.289,42.826,158.276
C08613=1040.187,332.276,-121.373,172.294,42.829,158.277
C08614=1040.195,332.524,-121.408,172.299,42.832,158.278
C08615=1040.202,332.771,-121.444,172.304,42.834,158.279
C08616=1040.209,333.019,-121.479,172.308,42.837,158.280
C08617=1040.217,333.267,-121.516,172.313,42.839,158.281
C08618=1040.224,333.513,-121.551,172.319,42.842,158.282
C08619=1040.234,333.863,-121.602,172.325,42.846,158.283
C08620=1040.245,334.212,-121.652,172.332,42.849,158.285
C08621=1040.255,334.562,-121.703,172.339,42.853,158.286
C08622=1040.266,334.912,-121.754,172.345,42.857,158.288
C08623=1040.273,335.160,-121.790,172.351,42.860,158.289
C08624=1040.280,335.407,-121.827,172.356,42.862,158.290
C08625=1040.287,335.655,-121.862,172.360,42.865,158.291
C08626=1040.294,335.902,-121.898,172.365,42.868,158.292
C08627=1040.302,336.149,-121.934,172.370,42.871,158.293
C08628=1040.309,336.397,-121.971,172.375,42.874,158.294
C08629=1040.316,336.643,-122.007,172.380,42.877,158.295
C08630=1040.324,336.891,-122.043,172.385,42.879,158.296
C08631=1040.331,337.138,-122.079,172.390,42.882,158.297
C08632=1040.338,337.385,-122.116,172.395,42.885,158.298
C08633=1040.345,337.633,-122.152,172.400,42.888,158.299
C08634=1040.352,337.880,-122.188,172.405,42.890,158.300
C08635=1040.360,338.127,-122.224,172.409,42.893,158.301
C08636=1040.367,338.374,-122.261,172.415,42.896,158.302
C08637=1040.375,338.622,-122.298,172.420,42.899,158.303
C08638=1040.382,338.868,-122.334,172.425,42.902,158.304
C08639=1040.390,339.116,-122.370,172.430,42.905,158.305
C08640=1040.397,339.364,-122.407,172.435,42.907,158.306
C08641=1040.404,339.611,-122.443,172.440,42.910,158.307
C08642=1040.412,339.857,-122.479,172.445,42.913,158.308
C08643=1040.419,340.105,-122.516,172.450,42.916,158.309
C08644=1040.426,340.352,-122.552,172.455,42.919,158.310
C08645=1040.434,340.600,-122.589,172.460,42.922,158.311
C08646=1040.442,340.847,-122.626,172.466,42.925,158.312
C08647=1040.448,341.094,-122.662,172.471,42.927,158.313
C08648=1040.456,341.341,-122.698,172.475,42.931,158.314
C08649=1040.464,341.588,-122.735,172.480,42.933,158.315
C08650=1040.471,341.836,-122.772,172.486,42.936,158.317
C08651=1040.479,342.083,-122.808,172.491,42.939,158.318
C08652=1040.486,342.330,-122.846,172.496,42.942,158.319
C08653=1040.493,342.577,-122.882,172.502,42.945,158.320
C08654=1040.500,342.824,-122.919,172.506,42.948,158.321
C08655=1040.508,343.072,-122.955,172.511,42.951,158.322
C08656=1040.515,343.319,-122.993,172.517,42.954,158.323
C08657=1040.523,343.566,-123.030,172.522,42.957,158.324
C08658=1040.530,343.813,-123.067,172.527,42.960,158.325
C08659=1040.538,344.060,-123.103,172.533,42.963,158.326
C08660=1040.545,344.308,-123.140,172.537,42.966,158.327
C08661=1040.553,344.555,-123.177,172.542,42.969,158.328
C08662=1040.560,344.801,-123.214,172.548,42.972,158.330
C08663=1040.567,345.048,-123.252,172.553,42.975,158.331
C08664=1040.574,345.296,-123.288,172.559,42.978,158.332
C08665=1040.582,345.543,-123.326,172.564,42.981,158.333
C08666=1040.590,345.790,-123.363,172.569,42.984,158.334
C08667=1040.597,346.037,-123.400,172.575,42.987,158.335
C08668=1040.604,346.285,-123.437,172.580,42.991,158.336
C08669=1040.612,346.531,-123.474,172.585,42.994,158.337
C08670=1040.619,346.779,-123.511,172.590,42.997,158.339
C08671=1040.627,347.025,-123.548,172.595,43.000,158.340
C08672=1040.634,347.273,-123.586,172.601,43.003,158.341
C08673=1040.642,347.520,-123.624,172.606,43.006,158.342
C08674=1040.650,347.767,-123.661,172.612,43.009,158.343
C08675=1040.660,348.113,-123.713,172.620,43.013,158.345
C08676=1040.670,348.459,-123.766,172.627,43.018,158.346
C08677=1040.681,348.805,-123.817,172.635,43.022,158.348
C08678=1040.692,349.152,-123.870,172.642,43.027,158.350
C08679=1040.700,349.398,-123.907,172.647,43.030,158.351
C08680=1040.708,349.646,-123.945,172.652,43.033,158.352
C08681=1040.715,349.893,-123.983,172.658,43.036,158.353
C08682=1040.722,350.140,-124.020,172.664,43.040,158.354
C08683=1040.730,350.387,-124.058,172.669,43.043,158.356
C08684=1040.738,350.634,-124.095,172.674,43.046,158.357
C08685=1040.745,350.881,-124.133,172.680,43.049,158.358
C08686=1040.752,351.128,-124.170,172.686,43.053,158.359
C08687=1040.760,351.375,-124.209,172.691,43.056,158.360
C08688=1040.767,351.622,-124.246,172.696,43.059,158.362
C08689=1040.775,351.870,-124.284,172.702,43.063,158.363
C08690=1040.782,352.116,-124.322,172.708,43.066,158.364
C08691=1040.790,352.364,-124.360,172.713,43.069,158.365
C08692=1040.798,352.610,-124.398,172.718,43.072,158.366
C08693=1040.806,352.857,-124.435,172.725,43.076,158.368
C08694=1040.813,353.104,-124.473,172.731,43.079,158.369
C08695=1040.821,353.352,-124.511,172.736,43.082,158.370
C08696=1040.829,353.598,-124.550,172.742,43.086,158.371
C08697=1040.836,353.845,-124.587,172.747,43.089,158.373
C08698=1040.843,354.092,-124.625,172.753,43.093,158.374
C08699=1040.851,354.340,-124.663,172.758,43.096,158.375
C08700=1040.859,354.586,-124.702,172.764,43.100,158.376
C08701=1040.867,354.833,-124.740,172.769,43.103,158.378
C08702=1040.874,355.080,-124.778,172.775,43.106,158.379
C08703=1040.882,355.327,-124.816,172.781,43.110,158.380
C08704=1040.891,355.574,-124.854,172.787,43.113,158.381
C08705=1040.898,355.821,-124.891,172.793,43.116,158.383
C08706=1040.906,356.068,-124.930,172.798,43.120,158.384
C08707=1040.913,356.315,-124.968,172.804,43.123,158.385
C08708=1040.921,356.561,-125.007,172.809,43.127,158.386
C08709=1040.929,356.809,-125.044,172.815,43.130,158.388
C08710=1040.936,357.056,-125.083,172.821,43.133,158.389
C08711=1040.944,357.303,-125.122,172.827,43.137,158.390
C08712=1040.951,357.550,-125.160,172.833,43.141,158.392
C08713=1040.960,357.797,-125.199,172.838,43.144,158.393
C08714=1040.967,358.043,-125.237,172.844,43.148,158.394
C08715=1040.975,358.291,-125.276,172.850,43.152,158.395
C08716=1040.983,358.537,-125.314,172.856,43.155,158.397
C08717=1040.991,358.784,-125.352,172.862,43.158,158.398
C08718=1040.999,359.031,-125.391,172.868,43.162,158.399
C08719=1041.006,359.278,-125.430,172.873,43.166,158.401
C08720=1041.013,359.525,-125.468,172.880,43.169,158.402
C08721=1041.022,359.772,-125.507,172.886,43.173,158.403
C08722=1041.029,360.018,-125.546,172.891,43.176,158.405
C08723=1041.038,360.265,-125.584,172.897,43.180,158.406
C08724=1041.046,360.512,-125.623,172.904,43.183,158.407
C08725=1041.053,360.759,-125.662,172.909,43.187,158.409
C08726=1041.061,361.006,-125.701,172.915,43.191,158.410
C08727=1041.069,361.252,-125.739,172.921,43.195,158.411
C08728=1041.077,361.500,-125.778,172.927,43.198,158.413
C08729=1041.085,361.747,-125.817,172.933,43.202,158.414
C08730=1041.092,361.993,-125.856,172.939,43.206,158.416
C08731=1041.103,362.345,-125.912,172.947,43.211,158.417
C08732=1041.115,362.698,-125.967,172.956,43.217,158.419
C08733=1041.126,363.049,-126.023,172.965,43.222,158.421
C08734=1041.137,363.402,-126.079,172.974,43.227,158.423
C08735=1041.145,363.649,-126.118,172.980,43.231,158.425
C08736=1041.153,363.895,-126.158,172.985,43.234,158.426
C08737=1041.161,364.142,-126.196,172.992,43.238,158.428
C08738=1041.168,364.389,-126.236,172.998,43.242,158.429
C08739=1041.177,364.635,-126.275,173.004,43.246,158.430
C08740=1041.184,364.882,-126.314,173.010,43.250,158.432
C08741=1041.192,365.129,-126.353,173.016,43.254,158.433
C08742=1041.200,365.375,-126.393,173.023,43.258,158.435
C08743=1041.208,365.623,-126.432,173.029,43.262,158.436
C08744=1041.216,365.870,-126.472,173.035,43.266,158.438
C08745=1041.223,366.115,-126.511,173.041,43.269,158.439
C08746=1041.231,366.362,-126.551,173.047,43.273,158.440
C08747=1041.240,366.609,-126.590,173.054,43.277,158.442
C08748=1041.247,366.856,-126.630,173.060,43.281,158.443
C08749=1041.256,367.102,-126.669,173.067,43.285,158.445
C08750=1041.263,367.349,-126.709,173.072,43.289,158.446
C08751=1041.272,367.596,-126.749,173.078,43.293,158.448
C08752=1041.280,367.843,-126.788,173.085,43.296,158.449
C08753=1041.288,368.089,-126.828,173.091,43.301,158.451
C08754=1041.296,368.336,-126.868,173.098,43.305,158.452
C08755=1041.304,368.583,-126.907,173.104,43.309,158.454
C08756=1041.312,368.830,-126.947,173.111,43.312,158.455
C08757=1041.320,369.076,-126.986,173.117,43.317,158.457
C08758=1041.328,369.323,-127.026,173.123,43.321,158.458
C08759=1041.337,369.570,-127.066,173.129,43.325,158.459
C08760=1041.344,369.817,-127.105,173.136,43.328,158.461
C08761=1041.353,370.063,-127.145,173.142,43.333,158.463
C08762=1041.361,370.310,-127.185,173.149,43.337,158.464
C08763=1041.369,370.556,-127.225,173.156,43.341,158.466
C08764=1041.377,370.803,-127.265,173.162,43.345,158.467
C08765=1041.385,371.050,-127.305,173.169,43.349,158.469
C08766=1041.393,371.296,-127.345,173.175,43.353,158.470
C08767=1041.401,371.543,-127.386,173.182,43.358,158.472
C08768=1041.409,371.789,-127.425,173.188,43.361,158.473
C08769=1041.417,372.036,-127.466,173.195,43.366,158.475
C08770=1041.425,372.283,-127.506,173.201,43.370,158.476
C08771=1041.433,372.529,-127.546,173.208,43.374,158.478
C08772=1041.441,372.775,-127.587,173.215,43.378,158.479
C08773=1041.450,373.022,-127.627,173.221,43.383,158.481
C08774=1041.458,373.269,-127.667,173.228,43.387,158.483
C08775=1041.466,373.516,-127.707,173.235,43.391,158.484
C08776=1041.474,373.762,-127.748,173.241,43.395,158.486
C08777=1041.482,374.008,-127.788,173.248,43.400,158.487
C08778=1041.491,374.255,-127.829,173.254,43.404,158.489
C08779=1041.498,374.502,-127.869,173.261,43.409,158.491
C08780=1041.507,374.748,-127.909,173.268,43.413,158.492
C08781=1041.515,374.994,-127.950,173.274,43.417,158.494
C08782=1041.524,375.241,-127.991,173.281,43.422,158.495
C08783=1041.532,375.488,-128.032,173.288,43.425,158.497
C08784=1041.540,375.734,-128.072,173.295,43.430,158.499
C08785=1041.548,375.980,-128.113,173.301,43.434,158.500
C08786=1041.556,376.227,-128.154,173.308,43.439,158.502
C08787=1041.569,376.599,-128.214,173.318,43.445,158.504
C08788=1041.581,376.971,-128.276,173.329,43.452,158.507
C08789=1041.595,377.343,-128.337,173.339,43.459,158.509
C08790=1041.607,377.714,-128.399,173.350,43.465,158.512
C08791=1041.615,377.961,-128.440,173.356,43.470,158.514
C08792=1041.624,378.208,-128.481,173.363,43.474,158.515
C08793=1041.632,378.454,-128.522,173.370,43.478,158.517
C08794=1041.641,378.701,-128.563,173.378,43.483,158.519
C08795=1041.649,378.947,-128.604,173.385,43.488,158.520
C08796=1041.657,379.194,-128.645,173.392,43.492,158.522
C08797=1041.666,379.440,-128.686,173.398,43.497,158.524
C08798=1041.674,379.686,-128.727,173.405,43.501,158.525
C08799=1041.682,379.932,-128.768,173.413,43.506,158.527
C08800=1041.691,380.179,-128.810,173.420,43.510,158.529
C08801=1041.699,380.425,-128.851,173.427,43.515,158.531
C08802=1041.708,380.672,-128.893,173.434,43.520,158.532
C08803=1041.716,380.918,-128.933,173.440,43.524,158.534
C08804=1041.724,381.165,-128.976,173.448,43.529,158.536
C08805=1041.732,381.410,-129.017,173.455,43.534,158.538
C08806=1041.741,381.657,-129.058,173.462,43.538,158.539
C08807=1041.749,381.903,-129.099,173.469,43.543,158.541
C08808=1041.758,382.149,-129.141,173.477,43.548,158.543
C08809=1041.766,382.397,-129.183,173.484,43.553,158.545
C08810=1041.774,382.642,-129.224,173.491,43.557,158.546
C08811=1041.783,382.889,-129.266,173.499,43.562,158.548
C08812=1041.792,383.135,-129.307,173.506,43.567,158.550
C08813=1041.800,383.381,-129.349,173.513,43.572,158.552
C08814=1041.809,383.627,-129.391,173.521,43.576,158.554
C08815=1041.817,383.874,-129.432,173.528,43.581,158.555
C08816=1041.826,384.121,-129.474,173.535,43.586,158.557
C08817=1041.834,384.367,-129.516,173.543,43.591,158.559
C08818=1041.843,384.613,-129.557,173.550,43.596,158.561
C08819=1041.852,384.860,-129.599,173.557,43.601,158.563
C08820=1041.861,385.106,-129.641,173.565,43.605,158.565
C08821=1041.869,385.351,-129.683,173.572,43.610,158.566
C08822=1041.877,385.598,-129.725,173.579,43.615,158.568
C08823=1041.886,385.844,-129.767,173.587,43.620,158.570
C08824=1041.895,386.090,-129.809,173.594,43.625,158.572
C08825=1041.904,386.337,-129.851,173.602,43.630,158.574
C08826=1041.912,386.583,-129.893,173.609,43.635,158.576
C08827=1041.922,386.829,-129.935,173.616,43.640,158.577
C08828=1041.931,387.075,-129.977,173.624,43.645,158.579
C08829=1041.939,387.322,-130.019,173.632,43.649,158.581
C08830=1041.948,387.568,-130.062,173.640,43.654,158.583
C08831=1041.957,387.814,-130.103,173.647,43.660,158.585
C08832=1041.966,388.061,-130.145,173.655,43.664,158.587
C08833=1041.974,388.307,-130.188,173.662,43.670,158.589
C08834=1041.983,388.553,-130.230,173.670,43.675,158.591
C08835=1041.992,388.799,-130.273,173.678,43.680,158.593
C08836=1042.001,389.045,-130.315,173.686,43.685,158.595
C08837=1042.009,389.292,-130.358,173.693,43.690,158.597
C08838=1042.019,389.537,-130.400,173.701,43.695,158.599
C08839=1042.027,389.784,-130.442,173.708,43.701,158.601
C08840=1042.036,390.030,-130.485,173.717,43.705,158.602
C08841=1042.045,390.276,-130.528,173.724,43.710,158.604
C08842=1042.053,390.522,-130.571,173.732,43.716,158.606
C08843=1042.064,390.824,-130.623,173.742,43.722,158.609
C08844=1042.075,391.127,-130.675,173.751,43.729,158.611
C08845=1042.086,391.430,-130.728,173.761,43.735,158.614
C08846=1042.097,391.733,-130.781,173.771,43.742,158.616
C08847=1042.109,392.082,-130.841,173.782,43.749,158.619
C08848=1042.122,392.431,-130.903,173.793,43.757,158.622
C08849=1042.135,392.780,-130.963,173.805,43.764,158.625
C08850=1042.148,393.129,-131.025,173.816,43.772,158.628
C08851=1042.156,393.375,-131.068,173.824,43.777,158.630
C08852=1042.165,393.621,-131.111,173.832,43.783,158.632
C08853=1042.173,393.867,-131.154,173.840,43.788,158.634
C08854=1042.183,394.114,-131.197,173.848,43.793,158.636
C08855=1042.192,394.359,-131.240,173.856,43.799,158.638
C08856=1042.201,394.605,-131.283,173.865,43.804,158.640
C08857=1042.211,394.851,-131.327,173.873,43.810,158.642
C08858=1042.219,395.097,-131.370,173.881,43.815,158.645
C08859=1042.228,395.344,-131.413,173.889,43.821,158.647
C08860=1042.237,395.589,-131.457,173.897,43.827,158.649
C08861=1042.246,395.835,-131.500,173.906,43.832,158.651
C08862=1042.256,396.081,-131.544,173.913,43.837,158.653
C08863=1042.265,396.326,-131.587,173.922,43.843,158.655
C08864=1042.274,396.573,-131.631,173.930,43.849,158.657
C08865=1042.283,396.819,-131.674,173.939,43.854,158.659
C08866=1042.292,397.065,-131.719,173.947,43.860,158.662
C08867=1042.300,397.311,-131.762,173.956,43.866,158.664
C08868=1042.310,397.557,-131.806,173.965,43.871,158.666
C08869=1042.319,397.802,-131.849,173.972,43.877,158.668
C08870=1042.328,398.048,-131.894,173.981,43.883,158.670
C08871=1042.337,398.294,-131.937,173.989,43.889,158.673
C08872=1042.347,398.540,-131.981,173.998,43.894,158.675
C08873=1042.356,398.786,-132.025,174.007,43.900,158.677
C08874=1042.365,399.031,-132.069,174.015,43.906,158.679
C08875=1042.375,399.277,-132.113,174.024,43.911,158.681
C08876=1042.384,399.524,-132.157,174.032,43.917,158.684
C08877=1042.393,399.769,-132.201,174.041,43.923,158.686
C08878=1042.402,400.015,-132.245,174.050,43.929,158.688
C08879=1042.412,400.261,-132.289,174.058,43.935,158.691
C08880=1042.421,400.507,-132.333,174.067,43.940,158.693
C08881=1042.430,400.753,-132.377,174.076,43.947,158.695
C08882=1042.440,400.998,-132.422,174.085,43.952,158.697
C08883=1042.449,401.244,-132.466,174.093,43.958,158.700
C08884=1042.458,401.491,-132.510,174.102,43.964,158.702
C08885=1042.467,401.736,-132.555,174.111,43.970,158.704
C08886=1042.476,401.982,-132.599,174.120,43.976,158.707
C08887=1042.486,402.228,-132.643,174.128,43.982,158.709
C08888=1042.495,402.474,-132.688,174.137,43.988,158.711
C08889=1042.505,402.719,-132.733,174.146,43.994,158.714
C08890=1042.515,402.965,-132.777,174.155,44.000,158.716
C08891=1042.523,403.211,-132.822,174.164,44.006,158.718
C08892=1042.533,403.457,-132.866,174.172,44.012,158.721
C08893=1042.543,403.703,-132.911,174.182,44.018,158.723
C08894=1042.552,403.948,-132.956,174.191,44.024,158.725
C08895=1042.561,404.195,-133.001,174.200,44.031,158.728
C08896=1042.571,404.440,-133.045,174.209,44.037,158.730
C08897=1042.580,404.686,-133.091,174.218,44.043,158.733
C08898=1042.589,404.931,-133.136,174.228,44.049,158.735
C08899=1042.598,405.144,-133.175,174.235,44.055,158.737
C08900=1042.606,405.356,-133.213,174.243,44.060,158.739
C08901=1042.614,405.570,-133.253,174.251,44.066,158.742
C08902=1042.622,405.782,-133.292,174.259,44.071,158.744
C08903=1042.631,405.995,-133.331,174.267,44.077,158.746
C08904=1042.639,406.207,-133.369,174.274,44.082,158.748
C08905=1042.647,406.420,-133.409,174.283,44.087,158.750
C08906=1042.655,406.631,-133.448,174.291,44.093,158.752
C08907=1042.666,406.878,-133.493,174.301,44.099,158.755
C08908=1042.675,407.124,-133.539,174.310,44.105,158.757
C08909=1042.684,407.369,-133.584,174.319,44.112,158.760
C08910=1042.694,407.614,-133.629,174.328,44.118,158.762
C08911=1042.704,407.860,-133.675,174.338,44.125,158.765
C08912=1042.714,408.106,-133.720,174.347,44.131,158.767
C08913=1042.723,408.351,-133.766,174.357,44.138,158.770
C08914=1042.733,408.597,-133.811,174.366,44.144,158.773
C08915=1042.742,408.843,-133.856,174.377,44.151,158.775
C08916=1042.753,409.089,-133.902,174.386,44.157,158.778
C08917=1042.762,409.334,-133.947,174.395,44.163,158.780
C08918=1042.772,409.580,-133.993,174.405,44.170,158.783
C08919=1042.782,409.825,-134.039,174.414,44.177,158.785
C08920=1042.791,410.071,-134.085,174.425,44.183,158.788
C08921=1042.802,410.317,-134.131,174.434,44.190,158.791
C08922=1042.811,410.562,-134.177,174.444,44.196,158.793
C08923=1042.822,410.808,-134.222,174.453,44.203,158.796
C08924=1042.832,411.054,-134.268,174.464,44.210,158.799
C08925=1042.841,411.299,-134.314,174.473,44.216,158.801
C08926=1042.852,411.544,-134.360,174.483,44.223,158.804
C08927=1042.862,411.790,-134.406,174.493,44.229,158.807
C08928=1042.872,412.035,-134.452,174.503,44.237,158.809
C08929=1042.882,412.281,-134.498,174.513,44.243,158.812
C08930=1042.892,412.527,-134.545,174.523,44.250,158.815
C08931=1042.902,412.772,-134.590,174.533,44.257,158.817
C08932=1042.912,413.018,-134.637,174.543,44.264,158.820
C08933=1042.922,413.264,-134.683,174.553,44.271,158.823
C08934=1042.931,413.508,-134.730,174.563,44.277,158.826
C08935=1042.941,413.754,-134.777,174.574,44.284,158.829
C08936=1042.952,414.000,-134.823,174.583,44.291,158.831
C08937=1042.962,414.245,-134.870,174.594,44.298,158.834
C08938=1042.971,414.490,-134.916,174.604,44.306,158.837
C08939=1042.981,414.736,-134.963,174.615,44.312,158.840
C08940=1042.992,414.981,-135.009,174.625,44.320,158.843
C08941=1043.002,415.226,-135.056,174.635,44.326,158.845
C08942=1043.012,415.472,-135.103,174.645,44.334,158.848
C08943=1043.022,415.718,-135.150,174.656,44.340,158.851
C08944=1043.032,415.963,-135.197,174.666,44.348,158.854
C08945=1043.043,416.208,-135.243,174.676,44.354,158.857
C08946=1043.053,416.454,-135.290,174.688,44.362,158.860
C08947=1043.063,416.699,-135.338,174.697,44.369,158.863
C08948=1043.073,416.945,-135.384,174.708,44.376,158.865
C08949=1043.084,417.190,-135.431,174.719,44.383,158.868
C08950=1043.094,417.435,-135.478,174.729,44.390,158.871
C08951=1043.105,417.680,-135.525,174.740,44.398,158.874
C08952=1043.115,417.926,-135.572,174.751,44.405,158.877
C08953=1043.126,418.172,-135.620,174.762,44.412,158.880
C08954=1043.136,418.417,-135.667,174.772,44.420,158.883
C08955=1043.146,418.662,-135.714,174.783,44.427,158.886
C08956=1043.156,418.908,-135.762,174.794,44.434,158.889
C08957=1043.167,419.152,-135.810,174.805,44.442,158.892
C08958=1043.177,419.398,-135.857,174.816,44.449,158.895
C08959=1043.186,419.615,-135.899,174.826,44.456,158.898
C08960=1043.196,419.831,-135.941,174.835,44.462,158.901
C08961=1043.205,420.048,-135.983,174.845,44.469,158.903
C08962=1043.214,420.264,-136.025,174.855,44.475,158.906
C08963=1043.223,420.481,-136.067,174.864,44.482,158.909
C08964=1043.232,420.697,-136.110,174.874,44.489,158.911
C08965=1043.242,420.913,-136.152,174.884,44.496,158.914
C08966=1043.251,421.130,-136.194,174.894,44.502,158.917
C08967=1043.262,421.375,-136.242,174.906,44.509,158.920
C08968=1043.272,421.621,-136.290,174.917,44.517,158.923
C08969=1043.283,421.866,-136.338,174.928,44.525,158.926
C08970=1043.294,422.111,-136.386,174.939,44.532,158.929
C08971=1043.305,422.356,-136.434,174.951,44.540,158.933
C08972=1043.315,422.601,-136.482,174.962,44.548,158.936
C08973=1043.326,422.846,-136.531,174.973,44.556,158.939
C08974=1043.336,423.092,-136.578,174.985,44.563,158.942
C08975=1043.347,423.337,-136.626,174.996,44.571,158.945
C08976=1043.358,423.581,-136.675,175.008,44.579,158.949
C08977=1043.369,423.826,-136.723,175.020,44.587,158.952
C08978=1043.380,424.072,-136.772,175.031,44.595,158.955
C08979=1043.391,424.317,-136.820,175.043,44.603,158.958
C08980=1043.401,424.562,-136.868,175.054,44.610,158.962
C08981=1043.412,424.807,-136.917,175.066,44.618,158.965
C08982=1043.423,425.052,-136.966,175.078,44.626,158.968
C08983=1043.434,425.297,-137.014,175.090,44.634,158.972
C08984=1043.444,425.542,-137.063,175.102,44.642,158.975
C08985=1043.456,425.787,-137.112,175.114,44.650,158.978
C08986=1043.467,426.032,-137.161,175.125,44.658,158.982
C08987=1043.477,426.278,-137.210,175.138,44.666,158.985
C08988=1043.488,426.522,-137.258,175.149,44.674,158.989
C08989=1043.500,426.766,-137.307,175.162,44.682,158.992
C08990=1043.510,427.011,-137.357,175.174,44.690,158.995
C08991=1043.521,427.257,-137.405,175.186,44.699,158.999
C08992=1043.533,427.502,-137.454,175.198,44.707,159.002
C08993=1043.543,427.747,-137.504,175.211,44.715,159.006
C08994=1043.555,427.991,-137.553,175.222,44.723,159.009
C08995=1043.566,428.236,-137.602,175.235,44.731,159.013
C08996=1043.577,428.481,-137.651,175.248,44.739,159.016
C08997=1043.588,428.726,-137.700,175.260,44.748,159.020
C08998=1043.599,428.971,-137.750,175.273,44.756,159.023
C08999=1043.610,429.216,-137.801,175.284,44.765,159.027
C09000=1043.622,429.461,-137.850,175.297,44.773,159.030
C09001=1043.633,429.706,-137.899,175.310,44.782,159.034
C09002=1043.644,429.950,-137.949,175.323,44.790,159.037
C09003=1043.655,430.195,-137.999,175.335,44.799,159.041
C09004=1043.666,430.440,-138.049,175.348,44.807,159.045
C09005=1043.678,430.685,-138.098,175.361,44.815,159.048
C09006=1043.689,430.929,-138.149,175.374,44.824,159.052
C09007=1043.701,431.173,-138.198,175.387,44.833,159.056
C09008=1043.711,431.419,-138.248,175.399,44.841,159.059
C09009=1043.723,431.664,-138.299,175.412,44.850,159.063
C09010=1043.735,431.908,-138.348,175.425,44.859,159.067
C09011=1043.746,432.152,-138.399,175.438,44.868,159.070
C09012=1043.758,432.397,-138.449,175.451,44.876,159.074
C09013=1043.768,432.642,-138.499,175.464,44.885,159.078
C09014=1043.780,432.887,-138.549,175.478,44.894,159.082
